// ---- 20_Product/10_BCF/11_Conv/10_Base/F_DeleteDestination.TcPOU
FUNCTION F_DeleteDestination : BOOL
(**************************************************************************************
 * 	Application		:	BoxControl Framework
 *	Revision		:	$Revision: 404529 $
 *	Revision date	:	$Date: 2018-04-23 08:21:38 +0200 (Mo., 23 Apr 2018) $
 *	Last changed by	:	$Author: b7bolm $
 *	URL				:	$URL: http://almscdc.swisslog.com/repo/SWPD/Development/BoxControlFramework/20_Release/trunk/01_Software/BCF/BCF/JumpStart/20_Product/10_App/10_Base/10_Lib/10_Conv/F_DeleteDestination.TcPOU $
 *
 *	Purpose			:	Request to delete a Destination in the TU data of a position.
 *						When the destination gets found - clear all other optional destinations.
 *
 * ------------------------------------------------------------------------------------
 *	Copyright Swisslog [IP AG], Switzerland. All rights reserved.
 * 
 * ------------------------------------------------------------------------------------
 *	
 * 	Revision History: 
 *
 * 	VERSION			DATE			INITIALS			DESCRIPTION
 *	0.1				01.01.2001		swl					Example
 *
 **************************************************************************************)
VAR_INPUT
	eFunctionNumber		: E_FunctionNumber; // Number of the function
	ZoneNumber			: INT; // Number of the zone in the function
END_VAR

VAR
	TU_DataIndex	: DINT; // TU-DataIndex
	Idx	  			: INT; // Index variable
END_VAR

// Initialize
F_DeleteDestination := FALSE;

// Get TU_DataIndex
TU_DataIndex := F_GetTU_DataIndex(
					eFunctionNumber := eFunctionNumber, // Position
					ZoneNumber := ZoneNumber); // Zone

// Check if the destination and the current position matches 
FOR Idx := 1 TO TU_DataTable[TU_DataIndex].DataSet.NumberOfDest DO
	IF TU_DataTable[TU_DataIndex].Destination[Idx].eFunctionNumber = eFunctionNumber
	   AND TU_DataTable[TU_DataIndex].Destination[Idx].ZoneNumber = ZoneNumber THEN
		// Destination found
		F_DeleteDestination := TRUE;
		EXIT;
	END_IF
END_FOR

// Destination was found - Delete all other optional destinations and update job present
IF F_DeleteDestination THEN
	// Clear destination table 
	MEMSET(destAddr := ADR(TU_DataTable[TU_DataIndex].Destination),fillByte := 0, n := SIZEOF(TU_DataTable[TU_DataIndex].Destination));
		
	// Reset number of destinations and reset JobPresent
	TU_DataTable[TU_DataIndex].DataSet.NumberOfDest := 0;
	TU_DataTable[TU_DataIndex].DataSet.JobPresent := FALSE;
END_IF

END_FUNCTION

// ---- 20_Product/10_BCF/11_Conv/11_Com/11_ITC/FB_ITC_ConveyorEmulation.TcPOU
FUNCTION_BLOCK FB_ITC_ConveyorEmulation IMPLEMENTS ITF_ITC_Emulation
(**************************************************************************************
 * 	Application		:	BoxControl Framework
 *	Revision		:	$Revision: 404529 $
 *	Revision date	:	$Date: 2018-04-23 08:21:38 +0200 (Mo., 23 Apr 2018) $
 *	Last changed by	:	$Author: b7bolm $
 *	URL				:	$URL: http://almscdc.swisslog.com/repo/SWPD/Development/BoxControlFramework/20_Release/trunk/01_Software/BCF/BCF/JumpStart/20_Product/11_Emu/11_Com/10_Lib/10_Conv/11_ITC/FB_ITC_CoveyorEmulation.TcPOU $
 *
 *	Purpose			:	ITC - Message Manager emulation.
 *						Represents the interface between the application and the 
 *						communication. Serves as abstract layer to ensure application
 *						independency.
 *
 * ------------------------------------------------------------------------------------
 *	Copyright Swisslog [IP AG], Switzerland. All rights reserved.
 * 
 * ------------------------------------------------------------------------------------
 *	
 * 	Revision History: 
 *
 * 	VERSION			DATE			INITIALS			DESCRIPTION
 *	0.1				01.01.2001		swl					Example
 *
 **************************************************************************************)
VAR
	fbDebugMsg			: FB_DebugMsg; // Debug instance
	DebugMsg			: T_MAXSTRING; // Debug msg
	TelegramPosition	: ST_PositionIdent; // Position
	TelegramElement		: E_ElementNumber; // Element
	TelegramGroup		: E_GroupNumber; // Group
	TelegramSubsystem	: BOOL; // Telegram for Subsystem
	TU_DataIndex		: DINT; // TU Data index
	eMsgType			: E_ITC_MsgTypeConv; // Message type conveyor
	
	Data				: ST_ITC_GeneralData; // General data
END_VAR

;

METHOD M_AddData : BOOL
(**************************************************************************************
 * 	Application		:	BoxControl Framework
 *	Revision		:	$Revision: 404529 $
 *	Revision date	:	$Date: 2018-04-23 08:21:38 +0200 (Mo., 23 Apr 2018) $
 *	Last changed by	:	$Author: b7bolm $
 *	URL				:	$URL: http://almscdc.swisslog.com/repo/SWPD/Development/BoxControlFramework/20_Release/trunk/01_Software/BCF/BCF/JumpStart/20_Product/11_Emu/11_Com/10_Lib/10_Conv/11_ITC/FB_ITC_CoveyorEmulation.TcPOU $
 *
 *	Purpose			:	Add data to the emulation system
 *
 * ------------------------------------------------------------------------------------
 *	Copyright Swisslog [IP AG], Switzerland. All rights reserved.
 * 
 * ------------------------------------------------------------------------------------
 *	
 * 	Revision History: 
 *
 * 	VERSION			DATE			INITIALS			DESCRIPTION
 *	0.1				01.01.2001		swl					Example
 *
 **************************************************************************************)
VAR_INPUT
	meChannelSrc	: E_MFCS_Channel;
	mMsgType		: INT;
	mpData			: PVOID;
	mLen			: UDINT;
END_VAR

// Translate type to enumeration
eMsgType := mMsgType;

// Go to corresponding type
CASE eMsgType OF
	(****************************************************
	  No Message type
	*****************************************************)	
	E_ITC_MsgTypeConv.NO_MESSAGE_TYPE:
		;
		
	(****************************************************
	  Add TU request
	*****************************************************)	
	E_ITC_MsgTypeConv.E_ADD_TU_REQUEST:
		// Process
		M_AddData := M_ProcessATQ(
						meChannelSrc := meChannelSrc,
						mpATQ		 := mpData,
						mLen		 := mLen);
		
	(****************************************************
	  Remove TU request
	*****************************************************)	
	E_ITC_MsgTypeConv.E_REMOVE_TU_REQUEST:
		// Process
		M_AddData := M_ProcessRTQ(
						meChannelSrc := meChannelSrc,
						mpRTQ		 := mpData,
						mLen		 := mLen);
	
	(****************************************************
	  Error request
	*****************************************************)	
	E_ITC_MsgTypeConv.E_ERROR_REQUEST:
		// Process
		M_AddData := M_ProcessERQ(
						meChannelSrc := meChannelSrc,
						mpERQ		 := mpData,
						mLen		 := mLen);
	
ELSE
	// Unknown type
	DebugMsg := 'Unknown message type received';
	fbDebugMsg.M_SendErrorMsg(mMessage := DebugMsg);		
END_CASE
END_METHOD

{attribute 'object_name' := 'M_CallITC_Service'}
METHOD M_CallITC_Service : BOOL
END_METHOD

METHOD PRIVATE M_ProcessATQ : BOOL
(**************************************************************************************
 * 	Application		:	BoxControl Framework
 *	Revision		:	$Revision: 404529 $
 *	Revision date	:	$Date: 2018-04-23 08:21:38 +0200 (Mo., 23 Apr 2018) $
 *	Last changed by	:	$Author: b7bolm $
 *	URL				:	$URL: http://almscdc.swisslog.com/repo/SWPD/Development/BoxControlFramework/20_Release/trunk/01_Software/BCF/BCF/JumpStart/20_Product/11_Emu/11_Com/10_Lib/10_Conv/11_ITC/FB_ITC_CoveyorEmulation.TcPOU $
 *
 *	Purpose			:	Add ATQ
 *
 * ------------------------------------------------------------------------------------
 *	Copyright Swisslog [IP AG], Switzerland. All rights reserved.
 * 
 * ------------------------------------------------------------------------------------
 *	
 * 	Revision History: 
 *
 * 	VERSION			DATE			INITIALS			DESCRIPTION
 *	0.1				01.01.2001		swl					Example
 *
 **************************************************************************************)
VAR_INPUT
	meChannelSrc		: E_MFCS_Channel; // Source communicaton channel
	mpATQ				: POINTER TO ST_ITC_ATQ; // Pointer to ATQ
	mLen				: UDINT; // Data length
END_VAR

VAR
	mrFunction		: REFERENCE TO FB_BaseObjectEmulation;
END_VAR

// Search position in registry
TelegramPosition := F_SearchFunctionPosition(Position := mpATQ^.Position);

// If a position and zone was found
IF TelegramPosition.eFunctionNumber > E_FunctionNumber.F_BEGIN_FUNCTION AND
   TelegramPosition.ZoneNumber > 0 THEN
   
   // Store reference of this position
   mrFunction REF= FunctionRegistryEmulation[TelegramPosition.eFunctionNumber].rFunction;
   
   // Check the reference from this position is valid
   IF __ISVALIDREF(mrFunction) THEN
	   
		// Get Data index from this position
		TU_DataIndex := F_GetTU_DataIndexEmulation(
							eFunctionNumber := TelegramPosition.eFunctionNumber,
							ZoneNumber		:= TelegramPosition.ZoneNumber);
		
		// If no data was found on this position
		IF TU_DataIndex = 0 THEN
			// Create a new set
			TU_DataIndex := F_InsertTU_DataEmulation(
								eFunctionNumber := TelegramPosition.eFunctionNumber,
								ZoneNumber 		:= TelegramPosition.ZoneNumber);
	
			// If a index could be created
			IF TU_DataIndex > 0 THEN
				TU_DataTableEmulation[TU_DataIndex].Label.ASCII := mpATQ^.Label;
				TU_DataTableEmulation[TU_DataIndex].Label.HashCode := F_CreateHashCode(mpATQ^.Label);
				TU_DataTableEmulation[TU_DataIndex].DataSet.Dimension.Weight := mpATQ^.Weight;
				TU_DataTableEmulation[TU_DataIndex].DataSet.Dimension.Length := mpATQ^.Length;
				TU_DataTableEmulation[TU_DataIndex].DataSet.Dimension.Height := mpATQ^.Height;
				TU_DataTableEmulation[TU_DataIndex].DataSet.Dimension.Width := mpATQ^.Width;
				TU_DataTableEmulation[TU_DataIndex].DataSet.LongSideLeading := mpATQ^.LongSideLeading;
				TU_DataTableEmulation[TU_DataIndex].DataSet.DataPresent := TRUE;
				
				// Prepare data
				Data.TU_DataIndex := TU_DataIndex;
				Data.ZoneNumber := TelegramPosition.ZoneNumber;
				
				M_ProcessToFunction(
					meFunctionNumber := TelegramPosition.eFunctionNumber,
					mZoneNumber 	 := TelegramPosition.ZoneNumber,
					meChannelSrc	 := meChannelSrc,
					mMsgType		 := E_ITC_MsgTypeConv.E_ADD_TU_REQUEST,
					mpData			 := ADR(Data),
					mLen			 := SIZEOF(Data));
			END_IF
		
		// Otherwise overwrite current index
		ELSIF TU_DataIndex > 0 THEN
			
			// Overwrite
			TU_DataTableEmulation[TU_DataIndex].Label.ASCII := mpATQ^.Label;
			TU_DataTableEmulation[TU_DataIndex].Label.HashCode := F_CreateHashCode(mpATQ^.Label);
			TU_DataTableEmulation[TU_DataIndex].DataSet.Dimension.Weight := mpATQ^.Weight;
			TU_DataTableEmulation[TU_DataIndex].DataSet.Dimension.Length := mpATQ^.Length;
			TU_DataTableEmulation[TU_DataIndex].DataSet.Dimension.Height := mpATQ^.Height;
			TU_DataTableEmulation[TU_DataIndex].DataSet.Dimension.Width := mpATQ^.Width;
			TU_DataTableEmulation[TU_DataIndex].DataSet.LongSideLeading := mpATQ^.LongSideLeading;
			TU_DataTableEmulation[TU_DataIndex].DataSet.DataPresent := TRUE;
		END_IF
		
		F_ITC_SendATR(
			eChannelSrc  := meChannelSrc, 
			PositionName := mpATQ^.Position, 
			eReturnCode  := E_ErrorConv.NO_ERROR_CODE);
	END_IF

// Unknown destination received 
ELSE
	// debug message: '11-000-0000-00-0,  unknown position addressed,  telegram = ATQ,  Position = 99-999-9999-99-9'
	DebugMsg:= '';
	DebugMsg:= CONCAT(DebugMsg, F_AddDividerToSisString(SubsystemRegistry.SubsystemName));
	DebugMsg:= CONCAT(DebugMsg, ',  unknown position addressed');
	DebugMsg:= CONCAT(DebugMsg, DebugTextBlocks.TELEGRAM);
	DebugMsg:= CONCAT(DebugMsg, 'ATQ');
	DebugMsg:= CONCAT(DebugMsg, DebugTextBlocks.POSITION);
	DebugMsg:= CONCAT(DebugMsg, F_AddDividerToSisString(Name:= mpATQ^.Position)  );
	fbDebugMsg.M_SendErrorMsg(mMessage := DebugMsg);

	// Reject telegram
	F_ITC_SendATR(
		eChannelSrc  := meChannelSrc, 
		PositionName := mpATQ^.Position, 
		eReturnCode  := E_ErrorConv.FUNCTIONNUMBER_UNKNOWN);
END_IF
END_METHOD

METHOD PRIVATE M_ProcessERQ : BOOL
(**************************************************************************************
 * 	Application		:	BoxControl Framework
 *	Revision		:	$Revision: 404529 $
 *	Revision date	:	$Date: 2018-04-23 08:21:38 +0200 (Mo., 23 Apr 2018) $
 *	Last changed by	:	$Author: b7bolm $
 *	URL				:	$URL: http://almscdc.swisslog.com/repo/SWPD/Development/BoxControlFramework/20_Release/trunk/01_Software/BCF/BCF/JumpStart/20_Product/11_Emu/11_Com/10_Lib/10_Conv/11_ITC/FB_ITC_CoveyorEmulation.TcPOU $
 *
 *	Purpose			:	Add ERR
 *
 * ------------------------------------------------------------------------------------
 *	Copyright Swisslog [IP AG], Switzerland. All rights reserved.
 * 
 * ------------------------------------------------------------------------------------
 *	
 * 	Revision History: 
 *
 * 	VERSION			DATE			INITIALS			DESCRIPTION
 *	0.1				01.01.2001		swl					Example
 *
 **************************************************************************************)
VAR_INPUT
	meChannelSrc		: E_MFCS_Channel; // Source communicaton channel
	mpERQ				: POINTER TO ST_ITC_ERQ; // Pointer to ERQ
	mLen				: UDINT; // Data length
END_VAR

// Try to find position in registry
TelegramPosition := F_SearchFunctionPosition(Position := mpERQ^.Position);

// Try to find element in registry
TelegramElement := F_SearchElementPosition(ElementName := mpERQ^.Position);

// Try to find group in registry
TelegramGroup := F_SearchGroupNumber(GroupName := mpERQ^.Position);

// Is it for the Subsystem
TelegramSubsystem := F_EqualSisNames(Name1 := SubsystemRegistry.SubsystemName,
                                     Name2 := mpERQ^.Position);

// If a position was found
IF TelegramPosition.eFunctionNumber > E_FunctionNumber.F_BEGIN_FUNCTION THEN
   
	M_ProcessToFunction(
		meFunctionNumber	:= TelegramPosition.eFunctionNumber, 
		mZoneNumber			:= TelegramPosition.ZoneNumber, 
		meChannelSrc		:= meChannelSrc, 
		mMsgType			:= E_ITC_MsgTypeConv.E_ERROR_REQUEST,
		mpData				:= mpERQ, 
		mLen				:= mLen);

// If a element was found
ELSIF TelegramElement > E_ElementNumber.E_BEGIN_ELEMENT THEN
   
	M_ProcessToElement(
		meElementNumber	:= TelegramElement, 
		meChannelSrc	:= meChannelSrc, 
		mMsgType		:= E_ITC_MsgTypeConv.E_ERROR_REQUEST,
		mpData			:= mpERQ, 
		mLen			:= mLen);

// If a group was found
ELSIF TelegramGroup > E_GroupNumber.G_BEGIN_GROUP THEN
   
	M_ProcessToGroup(
		meGroupNumber	:= TelegramGroup, 
		meChannelSrc	:= meChannelSrc, 
		mMsgType		:= E_ITC_MsgTypeConv.E_ERROR_REQUEST,
		mpData			:= mpERQ, 
		mLen			:= mLen);
		
// If it was for the Subsystem
ELSIF TelegramSubsystem THEN
   
	M_ProcessToSubsystem(
		meChannelSrc	:= meChannelSrc, 
		mMsgType		:= E_ITC_MsgTypeConv.E_ERROR_REQUEST,
		mpData			:= mpERQ, 
		mLen			:= mLen);
   
ELSE
	F_ITC_SendERR(
		eChannelSrc	:= meChannelSrc, 
		PositionName:= mpERQ^.Position, 
		Code		:= mpERQ^.Code, 
		eReturnCode	:= E_ErrorConv.WRONG_VALUE);
		
	// Unknown destination received 
	DebugMsg := CONCAT('M_ProcessERQ, Unknown position in Telegram: ', mpERQ^.Position);
	fbDebugMsg.M_SendErrorMsg(mMessage := DebugMsg);	
END_IF
END_METHOD

METHOD PRIVATE M_ProcessRTQ : BOOL
(**************************************************************************************
 * 	Application		:	BoxControl Framework
 *	Revision		:	$Revision: 404529 $
 *	Revision date	:	$Date: 2018-04-23 08:21:38 +0200 (Mo., 23 Apr 2018) $
 *	Last changed by	:	$Author: b7bolm $
 *	URL				:	$URL: http://almscdc.swisslog.com/repo/SWPD/Development/BoxControlFramework/20_Release/trunk/01_Software/BCF/BCF/JumpStart/20_Product/11_Emu/11_Com/10_Lib/10_Conv/11_ITC/FB_ITC_CoveyorEmulation.TcPOU $
 *
 *	Purpose			:	Add RTQ
 *
 * ------------------------------------------------------------------------------------
 *	Copyright Swisslog [IP AG], Switzerland. All rights reserved.
 * 
 * ------------------------------------------------------------------------------------
 *	
 * 	Revision History: 
 *
 * 	VERSION			DATE			INITIALS			DESCRIPTION
 *	0.1				01.01.2001		swl					Example
 *
 **************************************************************************************)
VAR_INPUT
	meChannelSrc		: E_MFCS_Channel; // Source communicaton channel
	mpRTQ				: POINTER TO ST_ITC_RTQ; // Pointer to RTQ
	mLen				: UDINT; // Data length
END_VAR

// Search position in registry
TelegramPosition := F_SearchFunctionPosition(Position := mpRTQ^.Position);

// If a position and zone was found
IF TelegramPosition.eFunctionNumber > E_FunctionNumber.F_BEGIN_FUNCTION AND
   TelegramPosition.ZoneNumber > 0 THEN
   
	// Prepare data
	Data.ZoneNumber := TelegramPosition.ZoneNumber;
	
	M_ProcessToFunction(
		meFunctionNumber := TelegramPosition.eFunctionNumber,
		mZoneNumber 	 := TelegramPosition.ZoneNumber,
		meChannelSrc	 := meChannelSrc,
		mMsgType		 := E_ITC_MsgTypeConv.E_REMOVE_TU_REQUEST,
		mpData			 := ADR(Data),
		mLen		     := SIZEOF(Data));

ELSE
	// Position not valid
	F_ITC_SendRTR(
		eChannelSrc	:= meChannelSrc, 
		PositionName:= mpRTQ^.Position, 
		eReturnCode	:= E_ErrorConv.WRONG_VALUE);
		
	// Unknown destination received 
	DebugMsg := CONCAT('M_ProcessRTQ, Unknown position in Telegram: ', mpRTQ^.Position);
	fbDebugMsg.M_SendErrorMsg(mMessage := DebugMsg);	
END_IF
END_METHOD

METHOD PRIVATE M_ProcessToElement : BOOL
(**************************************************************************************
 * 	Application		:	BoxControl Framework
 *	Revision		:	$Revision: 404529 $
 *	Revision date	:	$Date: 2018-04-23 08:21:38 +0200 (Mo., 23 Apr 2018) $
 *	Last changed by	:	$Author: b7bolm $
 *	URL				:	$URL: http://almscdc.swisslog.com/repo/SWPD/Development/BoxControlFramework/20_Release/trunk/01_Software/BCF/BCF/JumpStart/20_Product/11_Emu/11_Com/10_Lib/10_Conv/11_ITC/FB_ITC_CoveyorEmulation.TcPOU $
 *
 *	Purpose			:	ITC - Process message to element
 *
 * ------------------------------------------------------------------------------------
 *	Copyright Swisslog [IP AG], Switzerland. All rights reserved.
 * 
 * ------------------------------------------------------------------------------------
 *	
 * 	Revision History: 
 *
 * 	VERSION			DATE			INITIALS			DESCRIPTION
 *	0.1				01.01.2001		swl					Example
 *
 **************************************************************************************)
VAR_INPUT
	meElementNumber	: E_ElementNumber;
	meChannelSrc	: E_MFCS_Channel; // Source communicaton channel
	mMsgType		: INT; // msg type
	mpData			: PVOID; // data pointer
	mLen			: UDINT; // Data length
END_VAR

VAR
	mrefObject		: REFERENCE TO FB_BaseObjectEmulation; // Reference
END_VAR
// Initialize
M_ProcessToElement := TRUE;

// Check if ElementNumber is valid
IF meElementNumber > E_ElementNumber.E_BEGIN_ELEMENT AND 
   meElementNumber < E_ElementNumber.E_END_ELEMENT THEN
	// Set reference
	mrefObject REF= ElementRegistryEmulation[meElementNumber].rElement;
	
	// Check if reference is valid
	IF __ISVALIDREF(mrefObject) THEN
			// Forward message to corresponding object
		M_ProcessToElement := mrefObject.M_ITC_ProcessMsg(
								meChannelSrc := meChannelSrc, 
								mMsgType	 := mMsgType, 
								mpData		 := mpData,
								mLen	     := mLen); 
	END_IF	
END_IF
END_METHOD

METHOD PRIVATE M_ProcessToFunction : BOOL
(**************************************************************************************
 * 	Application		:	BoxControl Framework
 *	Revision		:	$Revision: 404529 $
 *	Revision date	:	$Date: 2018-04-23 08:21:38 +0200 (Mo., 23 Apr 2018) $
 *	Last changed by	:	$Author: b7bolm $
 *	URL				:	$URL: http://almscdc.swisslog.com/repo/SWPD/Development/BoxControlFramework/20_Release/trunk/01_Software/BCF/BCF/JumpStart/20_Product/11_Emu/11_Com/10_Lib/10_Conv/11_ITC/FB_ITC_CoveyorEmulation.TcPOU $
 *
 *	Purpose			:	ITC - Process message to function
 *
 * ------------------------------------------------------------------------------------
 *	Copyright Swisslog [IP AG], Switzerland. All rights reserved.
 * 
 * ------------------------------------------------------------------------------------
 *	
 * 	Revision History: 
 *
 * 	VERSION			DATE			INITIALS			DESCRIPTION
 *	0.1				01.01.2001		swl					Example
 *
 **************************************************************************************)
VAR_INPUT
	meFunctionNumber	: E_FunctionNumber; // Function number
	mZoneNumber			: INT; // Zone number
	meChannelSrc		: E_MFCS_Channel; // Source communicaton channel
	mMsgType		: INT; // msg type
	mpData			: PVOID; // data pointer
	mLen			: UDINT; // Data length
END_VAR

VAR
	mrefObject			: REFERENCE TO FB_BaseObjectEmulation; // Reference
END_VAR
// Initialize
M_ProcessToFunction := TRUE;

// If a valid function was found with a valid zone
IF 	meFunctionNumber > E_FunctionNumber.F_BEGIN_FUNCTION AND 
	meFunctionNumber < E_FunctionNumber.F_END_FUNCTION AND 
	mZoneNumber >= 0 AND mZoneNumber <= NUMBER_OF_ZONES_PER_FUNCTION THEN

	// Set reference 
	mrefObject REF= FunctionRegistryEmulation[meFunctionNumber].rFunction;
	
	// Check if reference is valid
	IF __ISVALIDREF(mrefObject) THEN

		// Call M_ITC_AddToBuffer
		M_ProcessToFunction := mrefObject.M_ITC_ProcessMsg(
								meChannelSrc := meChannelSrc, 
								mMsgType	 := mMsgType, 
								mpData		 := mpData,
								mLen		 := mLen); 
	END_IF
END_IF
END_METHOD

METHOD PRIVATE M_ProcessToGroup : BOOL
(**************************************************************************************
 * 	Application		:	BoxControl Framework
 *	Revision		:	$Revision: 404529 $
 *	Revision date	:	$Date: 2018-04-23 08:21:38 +0200 (Mo., 23 Apr 2018) $
 *	Last changed by	:	$Author: b7bolm $
 *	URL				:	$URL: http://almscdc.swisslog.com/repo/SWPD/Development/BoxControlFramework/20_Release/trunk/01_Software/BCF/BCF/JumpStart/20_Product/11_Emu/11_Com/10_Lib/10_Conv/11_ITC/FB_ITC_CoveyorEmulation.TcPOU $
 *
 *	Purpose			:	ITC - Process message to group
 *
 * ------------------------------------------------------------------------------------
 *	Copyright Swisslog [IP AG], Switzerland. All rights reserved.
 * 
 * ------------------------------------------------------------------------------------
 *	
 * 	Revision History: 
 *
 * 	VERSION			DATE			INITIALS			DESCRIPTION
 *	0.1				01.01.2001		swl					Example
 *
 **************************************************************************************)
VAR_INPUT
	meGroupNumber		: E_GroupNumber; // Groupnumber
	meChannelSrc		: E_MFCS_Channel; // Source communicaton channel
	mMsgType		: INT; // msg type
	mpData			: PVOID; // data pointer
	mLen			: UDINT; // Data length
END_VAR

VAR
	mrefObject			: REFERENCE TO FB_BaseObjectEmulation; // Reference
END_VAR
// Initialize
M_ProcessToGroup := TRUE;

// Check if GroupNumber is valid
IF meGroupNumber > E_GroupNumber.G_BEGIN_GROUP AND 
   meGroupNumber < E_GroupNumber.G_END_GROUP THEN
	// Set reference
	mrefObject REF= GroupRegistryEmulation[meGroupNumber].rGroup;
	
	// Check if reference is valid
	IF __ISVALIDREF(mrefObject) THEN
		
		// Send ITC-message to a specified group
		M_ProcessToGroup := mrefObject.M_ITC_ProcessMsg(
								meChannelSrc := meChannelSrc, 
								mMsgType	 := mMsgType, 
								mpData		 := mpData,
								mLen		 := mLen); 	
	END_IF
END_IF
END_METHOD

METHOD PRIVATE M_ProcessToSubsystem : BOOL
(**************************************************************************************
 * 	Application		:	BoxControl Framework
 *	Revision		:	$Revision: 404529 $
 *	Revision date	:	$Date: 2018-04-23 08:21:38 +0200 (Mo., 23 Apr 2018) $
 *	Last changed by	:	$Author: b7bolm $
 *	URL				:	$URL: http://almscdc.swisslog.com/repo/SWPD/Development/BoxControlFramework/20_Release/trunk/01_Software/BCF/BCF/JumpStart/20_Product/11_Emu/11_Com/10_Lib/10_Conv/11_ITC/FB_ITC_CoveyorEmulation.TcPOU $
 *
 *	Purpose			:	ITC - Process message to subsystem
 *
 * ------------------------------------------------------------------------------------
 *	Copyright Swisslog [IP AG], Switzerland. All rights reserved.
 * 
 * ------------------------------------------------------------------------------------
 *	
 * 	Revision History: 
 *
 * 	VERSION			DATE			INITIALS			DESCRIPTION
 *	0.1				01.01.2001		swl					Example
 *
 **************************************************************************************)
VAR_INPUT
	meChannelSrc		: E_MFCS_Channel; // Source communicaton channel
	mMsgType		: INT; // msg type
	mpData			: PVOID; // data pointer
	mLen			: UDINT; // Data length
END_VAR

VAR
	mrefObject			: REFERENCE TO FB_BaseObjectEmulation; // Reference
END_VAR
// Initialize
M_ProcessToSubsystem := TRUE;

// Set reference 
mrefObject REF= SubsystemRegistryEmulation.rSubsystem;

// Check if reference is valid
IF __ISVALIDREF(mrefObject) THEN
	// Call M_ITC_AddToBuffer
	M_ProcessToSubsystem := mrefObject.M_ITC_ProcessMsg(
								meChannelSrc := meChannelSrc, 
								mMsgType	 := mMsgType, 
								mpData		 := mpData,
								mLen		 := mLen);
END_IF
END_METHOD

END_FUNCTION_BLOCK

// ---- 20_Product/10_BCF/11_Conv/11_Com/11_ITC/F_ITC_SendATR.TcPOU
FUNCTION F_ITC_SendATR : BOOL
(**************************************************************************************
 * 	Application		:	BoxControl Framework
 *	Revision		:	$Revision: 404529 $
 *	Revision date	:	$Date: 2018-04-23 08:21:38 +0200 (Mo., 23 Apr 2018) $
 *	Last changed by	:	$Author: b7bolm $
 *	URL				:	$URL: http://almscdc.swisslog.com/repo/SWPD/Development/BoxControlFramework/20_Release/trunk/01_Software/BCF/BCF/JumpStart/20_Product/10_App/11_Com/10_Lib/10_Conv/11_ITC/F_ITC_SendATR.TcPOU $
 *
 *	Purpose			:	Wrap message - ATR
 *
 * ------------------------------------------------------------------------------------
 *	Copyright Swisslog [IP AG], Switzerland. All rights reserved.
 * 
 * ------------------------------------------------------------------------------------
 *	
 * 	Revision History: 
 *
 * 	VERSION			DATE			INITIALS			DESCRIPTION
 *	0.1				01.01.2001		swl					Example
 *
 **************************************************************************************)
VAR_INPUT
	eChannelSrc		: E_MFCS_Channel; // Source communicaton channel
	PositionName	: STRING(Conveyor.POSITION_STRINGLENGTH); // SIS MM-GGG-EEEE-FF-Z
	eReturnCode		: E_ErrorConv; // Return code
END_VAR
VAR
	ATR				: ST_ITC_ATR; 
END_VAR

// Map values
ATR.Position := PositionName;
ATR.ReturnCode := eReturnCode;

// Forward to ITC
F_ITC_SendATR := fbITC_Manager.M_SendData(
					meChannel	:= eChannelSrc,
					mMsgType	:= E_ITC_MsgTypeConv.E_ADD_TU_REPORT,
					mpData		:= ADR(ATR),
					mLen		:= SIZEOF(ATR));

END_FUNCTION

// ---- 20_Product/10_BCF/11_Conv/11_Com/11_ITC/F_ITC_SendERR.TcPOU
FUNCTION F_ITC_SendERR : BOOL
(**************************************************************************************
 * 	Application		:	BoxControl Framework
 *	Revision		:	$Revision: 404529 $
 *	Revision date	:	$Date: 2018-04-23 08:21:38 +0200 (Mo., 23 Apr 2018) $
 *	Last changed by	:	$Author: b7bolm $
 *	URL				:	$URL: http://almscdc.swisslog.com/repo/SWPD/Development/BoxControlFramework/20_Release/trunk/01_Software/BCF/BCF/JumpStart/20_Product/10_App/11_Com/10_Lib/10_Conv/11_ITC/F_ITC_SendERR.TcPOU $
 *
 *	Purpose			:	Wrap message - ERR
 *
 * ------------------------------------------------------------------------------------
 *	Copyright Swisslog [IP AG], Switzerland. All rights reserved.
 * 
 * ------------------------------------------------------------------------------------
 *	
 * 	Revision History: 
 *
 * 	VERSION			DATE			INITIALS			DESCRIPTION
 *	0.1				01.01.2001		swl					Example
 *
 **************************************************************************************)
VAR_INPUT
	eChannelSrc		: E_MFCS_Channel; // Source communicaton channel
	PositionName	: STRING(Conveyor.POSITION_STRINGLENGTH); // SIS MM-GGG-EEEE-FF-Z
	Code			: INT; // Error type code
	eReturnCode		: E_ErrorConv; // Return code
END_VAR
VAR
	ERR				: ST_ITC_ERR; 
END_VAR

// Map values
ERR.Position := PositionName;
ERR.Code := Code;
ERR.ReturnCode := eReturnCode;

// Forward to ITC
F_ITC_SendERR := fbITC_Manager.M_SendData(
					meChannel	:= eChannelSrc,
					mMsgType	:= E_ITC_MsgTypeConv.E_ERROR_REPORT,
					mpData		:= ADR(ERR),
					mLen		:= SIZEOF(ERR));

END_FUNCTION

// ---- 20_Product/10_BCF/11_Conv/11_Com/11_ITC/F_ITC_SendRTR.TcPOU
FUNCTION F_ITC_SendRTR : BOOL
(**************************************************************************************
 * 	Application		:	BoxControl Framework
 *	Revision		:	$Revision: 404529 $
 *	Revision date	:	$Date: 2018-04-23 08:21:38 +0200 (Mo., 23 Apr 2018) $
 *	Last changed by	:	$Author: b7bolm $
 *	URL				:	$URL: http://almscdc.swisslog.com/repo/SWPD/Development/BoxControlFramework/20_Release/trunk/01_Software/BCF/BCF/JumpStart/20_Product/10_App/11_Com/10_Lib/10_Conv/11_ITC/F_ITC_SendRTR.TcPOU $
 *
 *	Purpose			:	Wrap message - RTR
 *
 * ------------------------------------------------------------------------------------
 *	Copyright Swisslog [IP AG], Switzerland. All rights reserved.
 * 
 * ------------------------------------------------------------------------------------
 *	
 * 	Revision History: 
 *
 * 	VERSION			DATE			INITIALS			DESCRIPTION
 *	0.1				01.01.2001		swl					Example
 *
 **************************************************************************************)
VAR_INPUT
	eChannelSrc		: E_MFCS_Channel; // Source communicaton channel
	PositionName	: STRING(Conveyor.POSITION_STRINGLENGTH); // SIS MM-GGG-EEEE-FF-Z
	eReturnCode		: E_ErrorConv; // Return code
END_VAR
VAR
	RTR				: ST_ITC_RTR; 
END_VAR

// Map values
RTR.Position := PositionName;
RTR.ReturnCode := eReturnCode;

// Forward to ITC
F_ITC_SendRTR := fbITC_Manager.M_SendData(
					meChannel	:= eChannelSrc,
					mMsgType	:= E_ITC_MsgTypeConv.E_REMOVE_TU_REPORT,
					mpData		:= ADR(RTR),
					mLen		:= SIZEOF(RTR));

END_FUNCTION

// ---- 20_Product/20_ProBox/10_Base/09_Overrides/FB_PB_ITC_Conveyor.TcPOU
FUNCTION_BLOCK FB_PB_ITC_Conveyor EXTENDS FB_ITC_Conveyor IMPLEMENTS ITF_ITC 
(**************************************************************************************
 * 	Application		:	BoxControl Framework
 *	Revision		:	$Revision: 417092 $
 *	Revision date	:	$Date: 2018-11-14 12:58:58 +0100 (Mi., 14 Nov 2018) $
 *	Last changed by	:	$Author: q8aberh $
 *	URL				:	$URL: http://almscdc.swisslog.com/repo/SWPD/Development/ProMove/02_Controls/ProBox/03_Implementation/01_DevelopmentProject/01_Software/ProBox_COE/ProBox_DevProj_v1.0/PLC_1/20_Product/10_App/11_Com/10_Lib/10_Conv/11_ITC/FB_ITC_Conveyor.TcPOU $
 *
 *	Purpose			:	ITC - Message Manager.
 *						Represents the interface between the application and the 
 *						communication. Serves as abstract layer to ensure application
 *						independency.
 *
 * ------------------------------------------------------------------------------------
 *	Copyright Swisslog [IP AG], Switzerland. All rights reserved.
 * 
 * ------------------------------------------------------------------------------------
 *	
 * 	Revision History: 
 *
 * 	VERSION			DATE			INITIALS			DESCRIPTION
 *	0.1				01.01.2001		swl					Example
 *
 **************************************************************************************)
VAR_INPUT
	
END_VAR

VAR
	
END_VAR

VAR PERSISTENT
	
END_VAR

(**************************************************************************************************************
   Body never called!
***************************************************************************************************************)
;

METHOD PROTECTED M_ProcessTDQ : BOOL
(**************************************************************************************
 * 	Application		:	BoxControl Framework
 *	Revision		:	$Revision:  $
 *	Revision date	:	$Date: $
 *	Last changed by	:	$Author: q8hedls $
 *	URL				:	$URL: $
 *
 *	Purpose			:	Override BCF process for processing a received Task Delet Request telegram.
 *
 * ------------------------------------------------------------------------------------
 *	Copyright Swisslog [IP AG], Switzerland. All rights reserved.
 * 
 * ------------------------------------------------------------------------------------
 *	
 * 	Revision History: 
 *
 * 	VERSION			DATE			INITIALS			DESCRIPTION
 *	0.1				01.01.2001		swl					Example
 *
 **************************************************************************************)
VAR_INPUT
	meChannelSrc		: E_MFCS_Channel; // Source communicaton channel
	mpTDQ				: POINTER TO ST_ITC_TDQ; // Pointer to TDQ
	mLen				: UDINT; // Data length
END_VAR

VAR
	mPosition 			: ST_PositionIdent ; // Position
END_VAR

// Get position from telegram
mPosition := F_SearchFunctionPosition( Position := mpTDQ^.Position);
IF(mPosition.eFunctionNumber>E_FunctionNumber.F_BEGIN_FUNCTION AND mPosition.ZoneNumber>0) THEN
	F_ResetOccupied(mPosition.eFunctionNumber, mPosition.ZoneNumber);				
END_IF

//proceed with TDQ command
M_ProcessTDQ:= SUPER^.M_ProcessTDQ(meChannelSrc,mpTDQ,mLen);

//Re-initialize the function
IF(mPosition.eFunctionNumber>E_FunctionNumber.F_BEGIN_FUNCTION AND mPosition.ZoneNumber>0) THEN
	F_InitializeFunction(mPosition.eFunctionNumber);
END_IF
END_METHOD

METHOD PROTECTED M_ProcessTTA : BOOL
(**************************************************************************************
 * 	Application		:	BoxControl Framework
 *	Revision		:	$Revision:  $
 *	Revision date	:	$Date: $
 *	Last changed by	:	$Author: q8hedls $
 *	URL				:	$URL: $
 *
 *	Purpose			:	Override BCF process for processing a received Transport Task Assignment telegram.
 *
 * ------------------------------------------------------------------------------------
 *	Copyright Swisslog [IP AG], Switzerland. All rights reserved.
 * 
 * ------------------------------------------------------------------------------------
 *	
 * 	Revision History: 
 *
 * 	VERSION			DATE			INITIALS			DESCRIPTION
 *	0.1				01.01.2001		swl					Example
 *
 **************************************************************************************)
VAR_INPUT
	meChannelSrc		: E_MFCS_Channel; // Source communicaton channel
	mpTTA				: POINTER TO ST_ITC_TTA; // Pointer to TTA
	mLen				: UDINT;
END_VAR

VAR	
	mSensorOccupiedMem	: BOOL; //keep the actual value, to be able to set it back after the call to TTA cmd
	mRestore			: BOOL; //do a restore of SensorOccupied	
END_VAR

// Search position in registry
Position := F_SearchFunctionPosition(Position := mpTTA^.Position);
IF(__ISVALIDREF(F_PB_GetTransportControlDataRef(Position.eFunctionNumber, Position.ZoneNumber))) THEN
	mSensorOccupiedMem := F_PB_GetTransportControlDataRef(Position.eFunctionNumber, Position.ZoneNumber).SensorOccupied;
	mRestore := TRUE;
	IF(F_PB_GetTransportControlDataRef(Position.eFunctionNumber, Position.ZoneNumber).eTakeOverState <> E_TakeOverState.ACTIVE AND
	   F_PB_GetTransportControlDataRef(Position.eFunctionNumber, Position.ZoneNumber).eHandOverState <> E_HandOverState.ACTIVE) THEN
		//For Probox we want to be able to receive TTA despite there are not TU pressent, so we override the SensorOccupied value	   	
		F_PB_GetTransportControlDataRef(Position.eFunctionNumber, Position.ZoneNumber).SensorOccupied := TRUE;
	ELSE
		//force a TTC -> POSITION_NOT_CORRECT_OCCUPIED during an active transport.		
		F_PB_GetTransportControlDataRef(Position.eFunctionNumber, Position.ZoneNumber).SensorOccupied := FALSE;
	END_IF
END_IF
//proceed with TDQ command
M_ProcessTTA:= SUPER^.M_ProcessTTA(meChannelSrc,mpTTA,mLen);

//restore value
IF(mRestore) THEN
	F_PB_GetTransportControlDataRef(Position.eFunctionNumber, Position.ZoneNumber).SensorOccupied := mSensorOccupiedMem;
END_IF
END_METHOD

END_FUNCTION_BLOCK

// ---- 20_Product/20_ProBox/30_Toolbox/F_ResetOccupied.TcPOU
FUNCTION F_ResetOccupied : BOOL
(**************************************************************************************
 * 	Application		:	BoxControl Framework
 *	Revision		:	$Revision: 417092 $
 *	Revision date	:	$Date: 2018-11-14 12:58:58 +0100 (Mi., 14 Nov 2018) $
 *	Last changed by	:	$Author: q8aberh $
 *	URL				:	$URL: http://almscdc.swisslog.com/repo/SWPD/Development/ProMove/02_Controls/ProBox/03_Implementation/01_DevelopmentProject/01_Software/ProBox_COE/ProBox_DevProj_v1.0/PLC_1/20_Product/10_App/12_E_Functions/11_ProBox/02_Functions/F_ResetOccupied.TcPOU $
 *
 *	Purpose			:	Return zone data
 *
 * ------------------------------------------------------------------------------------
 *	Copyright Swisslog [IP AG], Switzerland. All rights reserved.
 * 
 * ------------------------------------------------------------------------------------
 *	
 * 	Revision History: 
 *
 * 	VERSION			DATE			INITIALS			DESCRIPTION
 *	0.1				01.01.2001		swl					Example
 *
 **************************************************************************************)
VAR_INPUT
	eFunctionNumber		: E_FunctionNumber;
	ZoneNumber			: INT; 
END_VAR



// Check if function number and zone is valid
IF eFunctionNumber > E_FunctionNumber.F_BEGIN_FUNCTION AND
   eFunctionNumber < E_FunctionNumber.F_END_FUNCTION AND
   ZoneNumber > 0 AND ZoneNumber <= NUMBER_OF_ZONES_PER_FUNCTION THEN
  
	// Check reference is valid
    IF __ISVALIDREF(FunctionRegistry[eFunctionNumber].rFunction) THEN
	   // Return zone data
	   //FunctionRegistry[eFunctionNumber].rFunction.M_DeleteOccupied(ZoneNumber);
	   IF __ISVALIDREF(FunctionRegistry[eFunctionNumber].Zone[ZoneNumber].refZoneData) THEN
		   FunctionRegistry[eFunctionNumber].Zone[ZoneNumber].refZoneData.TransportControlData.Occupied := FALSE;
		   FunctionRegistry[eFunctionNumber].Zone[ZoneNumber].refZoneData.TransportControlData.NumberOfPresentTUs := 0;
		   F_ResetOccupied := TRUE;
	   END_IF
    END_IF  
END_IF

END_FUNCTION

// ---- 20_Product/10_BCF/11_Conv/12_E_Functions/10_Helper/F_InitializeFunction.TcPOU
FUNCTION F_InitializeFunction :BOOL
(**************************************************************************************
 * 	Application		:	BoxControl Framework
 *	Revision		:	$Revision: 404529 $
 *	Revision date	:	$Date: 2018-04-23 08:21:38 +0200 (Mo., 23 Apr 2018) $
 *	Last changed by	:	$Author: b7bolm $
 *	URL				:	$URL: http://almscdc.swisslog.com/repo/SWPD/Development/BoxControlFramework/20_Release/trunk/01_Software/BCF/BCF/JumpStart/20_Product/10_App/12_E_Functions/10_Lib/10_Conv/10_Functions/F_InitializeFunction.TcPOU $
 *
 *	Purpose			:	Initialize all functions
 *
 * ------------------------------------------------------------------------------------
 *	Copyright Swisslog [IP AG], Switzerland. All rights reserved.
 * 
 * ------------------------------------------------------------------------------------
 *	
 * 	Revision History: 
 *
 * 	VERSION			DATE			INITIALS			DESCRIPTION
 *	0.1				01.01.2001		swl					Example
 *
 **************************************************************************************)
VAR_INPUT
	eFunctionNumber		: E_FunctionNumber; // Function number
END_VAR



// If reference is valid
IF __ISVALIDREF(FunctionRegistry[eFunctionNumber].rFunction) THEN
	// Initialize function
	FunctionRegistry[eFunctionNumber].rFunction.M_InitFunction(TRUE);
END_IF

END_FUNCTION

// ---- 20_Product/20_ProBox/30_Toolbox/F_PB_GetTransportControlDataRef.TcPOU
FUNCTION F_PB_GetTransportControlDataRef : REFERENCE TO ST_TransportControlData
(**************************************************************************************
 * 	Application		:	BoxControl Framework
 *	Revision		:	$Revision:  $
 *	Revision date	:	$Date: $
 *	Last changed by	:	$Author: q8sheds $
 *	URL				:	$URL: $
 *
 *	Purpose			:	return Transport control data as reference
 *
 * ------------------------------------------------------------------------------------
 *	Copyright Swisslog [IP AG], Switzerland. All rights reserved.
 * 
 * ------------------------------------------------------------------------------------
 *	
 * 	Revision History: 
 *
 * 	VERSION			DATE			INITIALS			DESCRIPTION
 *	0.1				01.01.2001		swl					Example
 *
 **************************************************************************************)
VAR_INPUT
	eFunctionNumber		: E_FunctionNumber; // Function number
	ZoneNumber			: INT; // Zone number
END_VAR

//init
F_PB_GetTransportControlDataRef REF= PBTransportCtrl.pbTransportControlDataEmpty;	//return ref to empty transportcontroller data to avoid reutrn of NULL

// Check if function number is valid
IF(  eFunctionNumber > E_FunctionNumber.F_BEGIN_FUNCTION AND eFunctionNumber < E_FunctionNumber.F_END_FUNCTION AND
	 ZoneNumber > 0 AND ZoneNumber <= NUMBER_OF_ZONES_PER_FUNCTION) THEN
	// Check reference is valid
	IF __ISVALIDREF(FunctionRegistry[eFunctionNumber].Zone[ZoneNumber].refZoneData) THEN
   		// Return transport control data   				
		F_PB_GetTransportControlDataRef REF= FunctionRegistry[eFunctionNumber].Zone[ZoneNumber].refZoneData.TransportControlData;
	END_IF
END_IF

END_FUNCTION

// ---- 20_Product/10_BCF/10_Base/10_StateMachine/FB_StateMachine.TcPOU
/// represents a state machine
{attribute 'no_explicit_call' := 'do not call this POU directly'} 
{attribute 'reflection'} 
FUNCTION_BLOCK PUBLIC FB_StateMachine
(**************************************************************************************
 *  Application     :   BoxControl Framework
 *  Revision date   :   $Date: 2021-04-09 08:29:02 +0200 (fre, 09 apr 2021) $
 *  Author          :   CDC
 * ------------------------------------------------------------------------------------
 *  © Swisslog AG
 *  Swisslog is not liable for any usage of this source code that is not agreed 
 *  on between Swisslog and the other party. The mandatory legal liability remains 
 *  unaffected.
 * ------------------------------------------------------------------------------------
 *  Revision History: 
 *
 *  VERSION DATE         INITIALS     DESCRIPTION
 *  0.0     DD.MM.YYYY   (name)       (explain customized modifications)
 *
 **************************************************************************************)
VAR
  {attribute 'instance-path'}
  {attribute 'no_init'}
  Instance          : STRING[255];     // instance path

  SisNbr            : A_InstancePath;  // SIS Number
  Name              : A_InstancePath;  // state machine name
  Tracing           : BOOL  := TRUE;   // HI = state changes are being traced

  State             : UINT;           // current state
  FStateChanged     : BOOL;           // state changed (and new state not yet arrived) 
  TimeStamp         : TIME;           // timestamp of state change
  Duration          : TIME;           // duration of last state

  Callback  : I_StateMachineTextCallback;	// callback event to retrieve state text

  Diagnose  : STRING[255];
END_VAR

VAR_STAT CONSTANT
  REASON_TEXT_LENGTH    : UINT          := 127;
  ARROW                 : STRING[7]     := ' => ';
  MISSING_CALLBACK		: A_StateText   := 'missing StateTextCallback';
END_VAR

METHOD FB_init : BOOL
(**************************************************************************************
 *  Application     :   BoxControl Framework
 *  Revision date   :   $Date: 2021-04-09 08:29:02 +0200 (fre, 09 apr 2021) $
 *  Author          :   CDC
 * ------------------------------------------------------------------------------------
 *  © Swisslog AG
 *  Swisslog is not liable for any usage of this source code that is not agreed 
 *  on between Swisslog and the other party. The mandatory legal liability remains 
 *  unaffected.
 * ------------------------------------------------------------------------------------
 *  Revision History: 
 *
 *  VERSION DATE         INITIALS     DESCRIPTION
 *  0.0     DD.MM.YYYY   (name)       (explain customized modifications)
 *
 **************************************************************************************)
VAR_INPUT
	bInitRetains		: BOOL; // if TRUE, the retain variables are initialized (warm start / cold start)
	bInCopyCode			: BOOL;  // if TRUE, the instance afterwards gets moved into the copy code (online change)

	mName				: A_InstancePath;       		// state machine name
	mStateTextCallback	: I_StateMachineTextCallback;	// callback event to retrieve state text
END_VAR

VAR
	SrcPos  : UINT;
	DstPos  : UINT;
	Length  : UINT;
END_VAR
Name        := mName;
Callback    := mStateTextCallback;

//Remove 'QB2Jumpstart.JumpStart.' from the instance path 
F_InstancePathRemovals(DestStart     := ADR(Instance),
                       DestEnd       := ADR(Instance) + SIZEOF(Instance),
                       RemoveLastPart:= FALSE );
END_METHOD

METHOD PROTECTED M_BuildTraceText
(**************************************************************************************
 *  Application     :   BoxControl Framework
 *  Revision date   :   $Date: 2021-04-09 08:29:02 +0200 (fre, 09 apr 2021) $
 *  Author          :   CDC
 * ------------------------------------------------------------------------------------
 *  © Swisslog AG
 *  Swisslog is not liable for any usage of this source code that is not agreed 
 *  on between Swisslog and the other party. The mandatory legal liability remains 
 *  unaffected.
 * ------------------------------------------------------------------------------------
 *  Revision History: 
 *
 *  VERSION DATE         INITIALS     DESCRIPTION
 *  0.0     DD.MM.YYYY   (name)       (explain customized modifications)
 *
 **************************************************************************************)
VAR_INPUT
  meMsgType       : E_DebugMsgType := E_DebugMsgType.INFO;
  mNewState      : UINT;
  mLastState     : UINT;
  mReason        : POINTER TO BYTE;
END_VAR

VAR
  Trace         : STRING[255];
  LastStateText : A_StateText := MISSING_CALLBACK;
  StateText     : A_StateText := MISSING_CALLBACK;
  DestStart     : POINTER TO BYTE;     // start position to concat
  DestEnd       : POINTER TO BYTE;     // buffer/string end
END_VAR
IF (Tracing = FALSE)
THEN
  RETURN;
END_IF

// get state texts
IF (Callback <> 0)
THEN
  LastStateText:= Callback.M_GetStateText(StateMachine:= THIS, StateNbr:= mLastState );
  StateText    := Callback.M_GetStateText(StateMachine:= THIS, StateNbr:=     P_State );
END_IF

// create trace text
DestStart:= ADR(Trace);
DestEnd  := ADR(Trace) + SIZEOF(Trace);
// sis nbr
DestStart:= F_StringCopy     (DestStart:= DestStart,  DestEnd:= DestEnd,  Source:= ADR(SisNbr)  );

// name
DestStart:= F_StringCopy     (DestStart:= DestStart,  DestEnd:= DestEnd,  Source:= ADR(',  ')  );
DestStart:= F_StringCopy     (DestStart:= DestStart,  DestEnd:= DestEnd,  Source:= ADR(Name)  );
DestStart:= F_StringCopy     (DestStart:= DestStart,  DestEnd:= DestEnd,  Source:= ADR(' changed')  );

// old state
DestStart:= F_StringCopy     (DestStart:= DestStart,  DestEnd:= DestEnd,  Source:= ADR(',  ')  );
DestStart:= F_StringFromUlint(DestStart:= DestStart,  DestEnd:= DestEnd,  Value := mLastState,  Length:= 0  );
DestStart:= F_StringCopy     (DestStart:= DestStart,  DestEnd:= DestEnd,  Source:= ADR(' (')  );
DestStart:= F_StringCopy     (DestStart:= DestStart,  DestEnd:= DestEnd,  Source:= ADR(LastStateText)  );
DestStart:= F_StringCopy     (DestStart:= DestStart,  DestEnd:= DestEnd,  Source:= ADR(')')  );

// new state
DestStart:= F_StringCopy     (DestStart:= DestStart,  DestEnd:= DestEnd,  Source:= ADR(ARROW)  );
DestStart:= F_StringFromUlint(DestStart:= DestStart,  DestEnd:= DestEnd,  Value := State,  Length:= 0  );
DestStart:= F_StringCopy     (DestStart:= DestStart,  DestEnd:= DestEnd,  Source:= ADR(' (')  );
DestStart:= F_StringCopy     (DestStart:= DestStart,  DestEnd:= DestEnd,  Source:= ADR(StateText)  );
DestStart:= F_StringCopy     (DestStart:= DestStart,  DestEnd:= DestEnd,  Source:= ADR(')')  );

// duration
DestStart:= F_StringCopy     (DestStart:= DestStart,  DestEnd:= DestEnd,  Source:= ADR(', duration = ')  );
DestStart:= F_StringFromTime (DestStart:= DestStart,  DestEnd:= DestEnd,  Value := Duration  );

// reason
DestStart:= F_StringCopy     (DestStart:= DestStart,  DestEnd:= DestEnd,  Source:= ADR(', reason = ')  );
DestStart:= F_StringCopy     (DestStart:= DestStart,  DestEnd:= DestEnd,  Source:= mReason  );

// to debug channel
fbDebugMsgManager.M_SendMessage(meMessageType:= meMsgType,
							  mDebugSource := Instance,
							  mpMsgData    := ADR(Trace),
							  mMsgDataLen  := DestStart - ADR(Trace) );

Diagnose:= Trace;
END_METHOD

/// returns the remaining time of state for the given duration
METHOD PUBLIC M_GetRemainingTime : TIME
(**************************************************************************************
 *  Application     :   BoxControl Framework
 *  Revision date   :   $Date: 2021-04-09 08:29:02 +0200 (fre, 09 apr 2021) $
 *  Author          :   CDC
 * ------------------------------------------------------------------------------------
 *  © Swisslog AG
 *  Swisslog is not liable for any usage of this source code that is not agreed 
 *  on between Swisslog and the other party. The mandatory legal liability remains 
 *  unaffected.
 * ------------------------------------------------------------------------------------
 *  Revision History: 
 *
 *  VERSION DATE         INITIALS     DESCRIPTION
 *  0.0     DD.MM.YYYY   (name)       (explain customized modifications)
 *
 **************************************************************************************)
VAR_INPUT
  mDuration  : TIME;    // total duration
END_VAR

VAR
  Remain    : TIME;
END_VAR
IF (P_TimeInState > mDuration)  THEN 
    Remain:= T#0S;
ELSE
    Remain:= mDuration - P_TimeInState;
END_IF

M_GetRemainingTime:= Remain;
END_METHOD

/// re entres the same state with reason
METHOD PUBLIC M_ReEntry
(**************************************************************************************
 *  Application     :   BoxControl Framework
 *  Revision date   :   $Date: 2021-04-09 08:29:02 +0200 (fre, 09 apr 2021) $
 *  Author          :   CDC
 * ------------------------------------------------------------------------------------
 *  © Swisslog AG
 *  Swisslog is not liable for any usage of this source code that is not agreed 
 *  on between Swisslog and the other party. The mandatory legal liability remains 
 *  unaffected.
 * ------------------------------------------------------------------------------------
 *  Revision History: 
 *
 *  VERSION DATE         INITIALS     DESCRIPTION
 *  0.0     DD.MM.YYYY   (name)       (explain customized modifications)
 *
 **************************************************************************************)
VAR_INPUT
  mReason                : STRING[REASON_TEXT_LENGTH]       := '';
END_VAR
FStateChanged:= TRUE;
Duration     := F_GetTimeMsDiff(TimeStamp);
TimeStamp    := F_GetTimeMsTick();


M_BuildTraceText(meMsgType  := E_DebugMsgType.INFO,
                 mNewState := State,
                 mLastState:= State,
                 mReason   := ADR(mReason)  );
END_METHOD

/// sets a new state with reason for change
METHOD PUBLIC M_SetState
(**************************************************************************************
 *  Application     :   BoxControl Framework
 *  Revision date   :   $Date: 2021-04-09 08:29:02 +0200 (fre, 09 apr 2021) $
 *  Author          :   CDC
 * ------------------------------------------------------------------------------------
 *  © Swisslog AG
 *  Swisslog is not liable for any usage of this source code that is not agreed 
 *  on between Swisslog and the other party. The mandatory legal liability remains 
 *  unaffected.
 * ------------------------------------------------------------------------------------
 *  Revision History: 
 *
 *  VERSION DATE         INITIALS     DESCRIPTION
 *  0.0     DD.MM.YYYY   (name)       (explain customized modifications)
 *
 **************************************************************************************)
VAR_INPUT
  mState     : UINT;
  mReason    : STRING[REASON_TEXT_LENGTH];
END_VAR

VAR
  LastState : UINT;
END_VAR
IF State = mState
THEN
  RETURN;
END_IF

LastState:= State;
State   :=  mState;

FStateChanged:= TRUE;
Duration     := F_GetTimeMsDiff(TimeStamp);
TimeStamp    := F_GetTimeMsTick();


M_BuildTraceText(meMsgType  := E_DebugMsgType.INFO,
                 mNewState := State,
                 mLastState:= LastState,
                 mReason   := ADR(mReason)  );
END_METHOD

/// sets a new state with reason for change and severity
METHOD PUBLIC M_SetState1
(**************************************************************************************
 *  Application     :   BoxControl Framework
 *  Revision date   :   $Date: 2021-04-09 08:29:02 +0200 (fre, 09 apr 2021) $
 *  Author          :   CDC
 * ------------------------------------------------------------------------------------
 *  © Swisslog AG
 *  Swisslog is not liable for any usage of this source code that is not agreed 
 *  on between Swisslog and the other party. The mandatory legal liability remains 
 *  unaffected.
 * ------------------------------------------------------------------------------------
 *  Revision History: 
 *
 *  VERSION DATE         INITIALS     DESCRIPTION
 *  0.0     DD.MM.YYYY   (name)       (explain customized modifications)
 *
 **************************************************************************************)
VAR_INPUT
  mMsgType   : E_DebugMsgType := E_DebugMsgType.INFO;
  mState     : UINT;
  mReason    : STRING[REASON_TEXT_LENGTH];
END_VAR

VAR
  LastState : UINT;
END_VAR
IF State = mState
THEN
  RETURN;
END_IF

LastState:= State;
State   :=  mState;

FStateChanged:= TRUE;
Duration     := F_GetTimeMsDiff(TimeStamp);
TimeStamp    := F_GetTimeMsTick();


M_BuildTraceText(meMsgType  := mMsgType,
                 mNewState := State,
                 mLastState:= LastState,
                 mReason   := ADR(mReason)  );
END_METHOD

// entry into new state (must be checked)
//{attribute 'monitoring' := 'call'} no call here
PROPERTY PUBLIC P_Entering : BOOL
GET

(**************************************************************************************************************)
(**************************************************************************************************************)
IF ( FStateChanged = FALSE )
THEN
  P_Entering:= FALSE;
  RETURN;
END_IF




(**************************************************************************************************************)
(**************************************************************************************************************)
FStateChanged:= FALSE;




(**************************************************************************************************************)
(** done ******************************************************************************************************)
P_Entering := TRUE;
END_GET
END_PROPERTY

// exit from old state (optionally)
{attribute 'monitoring' := 'call'}
PROPERTY PUBLIC P_Exiting : BOOL
GET
P_Exiting:= FStateChanged;
END_GET
END_PROPERTY

// SisNbr to trace
{attribute 'monitoring' := 'call'}
PROPERTY PUBLIC P_SisNbr : A_InstancePath
GET
P_SisNbr:= SisNbr;
END_GET
SET
SisNbr:= P_SisNbr;
END_SET
END_PROPERTY

// current state as UINT
{attribute 'monitoring' := 'call'}
PROPERTY PUBLIC P_State : UINT
GET
P_State:= State;
END_GET
END_PROPERTY

// duration of this state
{attribute 'monitoring' := 'call'}
PROPERTY PUBLIC P_TimeInState : TIME
GET
P_TimeInState:= F_GetTimeMsDiff( TimeStamp );
END_GET
END_PROPERTY

// HI = state changes are being traced
{attribute 'monitoring' := 'call'}
PROPERTY PUBLIC P_Tracing : BOOL
GET
P_Tracing:= Tracing;
END_GET
SET
Tracing:= P_Tracing;
END_SET
END_PROPERTY

END_FUNCTION_BLOCK

// ---- 20_Product/10_BCF/10_Base/11_Com/01_Stringhandling/F_StringFromUlint.TcPOU
// converts word to string with specific length (adds zeros)
FUNCTION PUBLIC F_StringFromUlint : POINTER TO BYTE

(**************************************************************************************
 * 	Application		:	BoxControl Framework
 *	Revision		  :	$Revision: 461868 $
 *	Revision date	:	$Date: 1979-01-09 14:35:13 +0200 (Di., 09 Jan 1979) $
 *	Last changed by	:	$Author: b7lipim $
 *	URL				:	$URL: http://almscdc.swisslog.com/repo/SWPD/Development/BoxControlFramework/20_Release/branches/R1.x/01_Software/BCF/BCF/JumpStart/20_Product/10_BCF/10_Base/11_Com/12_DebugMsg/00_GVLs/DebugTextBlocks.TcGVL $
 *
 * ------------------------------------------------------------------------------------
 *	Copyright Swisslog [IP AG], Switzerland. All rights reserved.
 * 
 * ------------------------------------------------------------------------------------
 *	
 * 	Revision History: 
 *
 * VERSION DATE         INITIALS     DESCRIPTION
 * 0.0     DD.MM.YYYY   (name)       (explain customized modifications)
 *
 **************************************************************************************)

(********************************************************************************************************************************)
VAR_INPUT
  DestStart             : POINTER TO BYTE                  := 0;     // = ADR(MyString)                    -> start position to concat
  DestEnd               : POINTER TO BYTE                  := 0;     // = ADR(MyString) + SIZEOF(MyString) -> buffer/string end
  (*----------------------------------------------------------------------------------------------------------------------------*)
  Value                 : ULINT                            := 0;     // value to convert
  Length                : BYTE                             := 0;     // minimum string length (may be left stuffed with zeros)
END_VAR

(********************************************************************************************************************************)
VAR
  DestWork              : POINTER TO BYTE                  := 0;
  (*----------------------------------------------------------------------------------------------------------------------------*)
  Result                : STRING[63]                       := '';
  Size                  : WORD                             := 0;
  Stuff                 : WORD                             := 0;
END_VAR


(********************************************************************************************************************************)
(** check inputs ****************************************************************************************************************)
IF   (DestStart = 0)         THEN  F_StringFromUlint:= 0;          RETURN;
ELSIF(DestEnd   = 0)         THEN  F_StringFromUlint:= DestStart;  RETURN;
ELSIF(DestStart >= DestEnd)  THEN  F_StringFromUlint:= DestStart;  RETURN;
END_IF

DestWork:= DestStart;




(********************************************************************************************************************************)
(** convert *********************************************************************************************************************)
Result:= ULINT_TO_STRING(Value);
Size  := INT_TO_WORD( LEN(Result) );




(********************************************************************************************************************************)
(** stuff? **********************************************************************************************************************)
IF (Size < Length)
THEN
  Stuff:= Length - Size;
  (*-----------------------------------------------------------------*)
  WHILE(Stuff > 0)
  DO
    Stuff:= Stuff - 1;
    (*-------------------------------------------*)
    IF (DestWork >= DestEnd)
    THEN
      DestWork := DestEnd - SIZEOF(DestWork^); // _DestWork^ hier benutzen
      DestWork^:= 16#00;
      DestWork := DestEnd;
      EXIT;
    END_IF
    (*-- add '0' --------------------------------*)
    DestWork^:= 16#30;
    DestWork := DestWork + SIZEOF(DestWork^);
  END_WHILE
END_IF




(********************************************************************************************************************************)
(** copy characters *************************************************************************************************************)
DestWork:= F_StringCopy( DestStart:= DestWork,
                         DestEnd  := DestEnd,
                         Source   := ADR(Result)  );




(********************************************************************************************************************************)
(** done ************************************************************************************************************************)
F_StringFromUlint:= DestWork;

END_FUNCTION

// ---- 20_Product/10_BCF/10_Base/11_Com/01_Stringhandling/F_StringFromTime.TcPOU
// converts word to string with specific length (adds zeros)
FUNCTION PUBLIC F_StringFromTime : POINTER TO BYTE

(**************************************************************************************
 * 	Application		:	BoxControl Framework
 *	Revision		  :	$Revision: 461868 $
 *	Revision date	:	$Date: 1979-01-09 14:35:13 +0200 (Di., 09 Jan 1979) $
 *	Last changed by	:	$Author: b7lipim $
 *	URL				:	$URL: http://almscdc.swisslog.com/repo/SWPD/Development/BoxControlFramework/20_Release/branches/R1.x/01_Software/BCF/BCF/JumpStart/20_Product/10_BCF/10_Base/11_Com/12_DebugMsg/00_GVLs/DebugTextBlocks.TcGVL $
 *
 * ------------------------------------------------------------------------------------
 *	Copyright Swisslog [IP AG], Switzerland. All rights reserved.
 * 
 * ------------------------------------------------------------------------------------
 *	
 * 	Revision History: 
 *
 * VERSION DATE         INITIALS     DESCRIPTION
 * 0.0     DD.MM.YYYY   (name)       (explain customized modifications)
 *
 **************************************************************************************)

(********************************************************************************************************************************)
VAR_INPUT
  DestStart             : POINTER TO BYTE                  := 0;     // = ADR(MyString)                    -> start position to concat
  DestEnd               : POINTER TO BYTE                  := 0;     // = ADR(MyString) + SIZEOF(MyString) -> buffer/string end
  (*----------------------------------------------------------------------------------------------------------------------------*)
  Value                 : TIME                             := T#0S;  // value to convert
END_VAR

(********************************************************************************************************************************)
VAR
  DestWork              : POINTER TO BYTE                  := 0;
  (*----------------------------------------------------------------------------------------------------------------------------*)
  Result                : STRING[15]                       := '';
END_VAR


(********************************************************************************************************************************)
(** check inputs ****************************************************************************************************************)
IF   (DestStart = 0)         THEN  F_StringFromTime:= 0;          RETURN;
ELSIF(DestEnd   = 0)         THEN  F_StringFromTime:= DestStart;  RETURN;
ELSIF(DestStart >= DestEnd)  THEN  F_StringFromTime:= DestStart;  RETURN;
END_IF

DestWork:= DestStart;




(********************************************************************************************************************************)
(** convert *********************************************************************************************************************)
Result:= TIME_TO_STRING(Value);




(********************************************************************************************************************************)
(** copy characters *************************************************************************************************************)
DestWork:= F_StringCopy( DestStart:= DestWork,
                         DestEnd  := DestEnd,
                         Source   := ADR(Result)  );




(********************************************************************************************************************************)
(** done ************************************************************************************************************************)
F_StringFromTime:= DestWork;

END_FUNCTION

// ---- 20_Product/10_BCF/10_Base/11_Com/02_Timings/F_GetBlinkCycle.TcPOU
// returns synchronized blinking pulses with requested (discreet) frequency
FUNCTION PUBLIC F_GetBlinkCycle : BOOL

(**************************************************************************************
 * 	Application		:	BoxControl Framework
 *	Revision		  :	$Revision: 461868 $
 *	Revision date	:	$Date: 1979-01-09 14:35:13 +0200 (Di., 09 Jan 1979) $
 *	Last changed by	:	$Author: b7lipim $
 *	URL				:	$URL: http://almscdc.swisslog.com/repo/SWPD/Development/BoxControlFramework/20_Release/branches/R1.x/01_Software/BCF/BCF/JumpStart/20_Product/10_BCF/10_Base/11_Com/12_DebugMsg/00_GVLs/DebugTextBlocks.TcGVL $
 *
 * ------------------------------------------------------------------------------------
 *	Copyright Swisslog [IP AG], Switzerland. All rights reserved.
 * 
 * ------------------------------------------------------------------------------------
 *	
 * 	Revision History: 
 *
 * VERSION DATE         INITIALS     DESCRIPTION
 * 0.0     DD.MM.YYYY   (name)       (explain customized modifications)
 *
 **************************************************************************************)

(************************************************************************************************************)
VAR_INPUT
  BlinkFrequency        : E_BlinkFrequencies               := E_BlinkFrequencies.Off;
END_VAR

(************************************************************************************************************)
VAR
  {attribute 'displaymode':='hex'}  _TimeTick    : DWORD   := 0;
  {attribute 'displaymode':='hex'}  _TimeMask    : DWORD   := 0;
END_VAR


(********************************************************************************************************************************)
(** calculate *******************************************************************************************************************)
_TimeTick:= TIME_TO_DWORD( TIME() );
_TimeMask:= ( BlinkFrequency AND _TimeTick );




(********************************************************************************************************************************)
(** done ************************************************************************************************************************)
F_GetBlinkCycle:= ( _TimeMask <> 0 );

END_FUNCTION

// ---- 20_Product/10_BCF/10_Base/11_Com/02_Timings/F_GetTimeRemain.TcPOU
// returns remaining time from a timestamp to specified duration
FUNCTION PUBLIC F_GetTimeRemain : TIME

(**************************************************************************************
 * 	Application		:	BoxControl Framework
 *	Revision		  :	$Revision: 461868 $
 *	Revision date	:	$Date: 1979-01-09 14:35:13 +0200 (Di., 09 Jan 1979) $
 *	Last changed by	:	$Author: b7lipim $
 *	URL				:	$URL: http://almscdc.swisslog.com/repo/SWPD/Development/BoxControlFramework/20_Release/branches/R1.x/01_Software/BCF/BCF/JumpStart/20_Product/10_BCF/10_Base/11_Com/12_DebugMsg/00_GVLs/DebugTextBlocks.TcGVL $
 *
 * ------------------------------------------------------------------------------------
 *	Copyright Swisslog [IP AG], Switzerland. All rights reserved.
 * 
 * ------------------------------------------------------------------------------------
 *	
 * 	Revision History: 
 *
 * VERSION DATE         INITIALS     DESCRIPTION
 * 0.0     DD.MM.YYYY   (name)       (explain customized modifications)
 *
 **************************************************************************************)

(********************************************************************************************************************************)
VAR_INPUT
  Duration              : TIME                             := T#0S;    // total duration
  Timestamp             : TIME                             := T#0S;    // time stamp when started
END_VAR

(********************************************************************************************************************************)
VAR
  Elapsed               : TIME                             := T#0S;
  Remain                : TIME                             := T#0S;
END_VAR


(********************************************************************************************************************************)
(** calculate *******************************************************************************************************************)
Elapsed:= F_GetTimeMsDiff(Timestamp);

IF (Elapsed > Duration)  THEN  Remain:= T#0S;
ELSE                           Remain:= Duration - Elapsed;
END_IF



(********************************************************************************************************************************)
(** done ************************************************************************************************************************)
F_GetTimeRemain:= Remain;

END_FUNCTION

// ---- 20_Product/10_BCF/10_Base/F_MemStringReplace.TcPOU
FUNCTION F_MemStringReplace : BOOL
(**************************************************************************************
 * 	Application		:	BoxControl Framework
 *	Revision		:	$Revision: 404529 $
 *	Revision date	:	$Date: 2018-04-23 08:21:38 +0200 (Mo., 23 Apr 2018) $
 *	Last changed by	:	$Author: b7bolm $
 *	URL				:	$URL: http://almscdc.swisslog.com/repo/SWPD/Development/BoxControlFramework/20_Release/trunk/01_Software/BCF/BCF/JumpStart/20_Product/10_App/10_Base/10_Lib/F_MemStringReplace.TcPOU $
 *
 *	Purpose			:	Search in a pointer based structure for a find string, replace 
 *						it with replacement string. If replacement string is shorter, 
 *						move data to close the gap and clean last digits after movement.
 *
 *
 * ------------------------------------------------------------------------------------
 *	Copyright Swisslog [IP AG], Switzerland. All rights reserved.
 * 
 * ------------------------------------------------------------------------------------
 *	
 * 	Revision History: 
 *
 * 	VERSION			DATE			INITIALS			DESCRIPTION
 *	0.1				01.01.2001		swl					Example
 *
 **************************************************************************************)
VAR_INPUT
	pSrc 			: PVOID; // Pointer to source
	FindString		: STRING(MAX_DIGITS); // Find string
	Replacement 	: STRING(MAX_DIGITS); // Replacement string
END_VAR
VAR_IN_OUT
	SrcLen 			: UDINT; // Length of source structure
END_VAR
VAR
	Idx 			: UDINT; // Iterator
	ReplacmentLen 	: UDINT; // Length of string
	FindLen			: UDINT; // Length of string
	RelativeSrc		: UDINT; // Relative source pointer to close gap in data
	RelativeDest	: UDINT; // Relative destination pointer to close gap in data
	pFirstDataByte 	: POINTER TO BYTE; // Pointer to a byte
	pFirstFindByte	: POINTER TO BYTE; // Pointer to a byte
	byte1 			: BYTE;
	byte2			: BYTE;
END_VAR

VAR CONSTANT
	MAX_DIGITS : UDINT := 10; // Max Digits of strings
END_VAR

(* 
Validate Inputs

Length of replacement needs to have the same or a smaller length,
compared to find. Otherwise it would be possible to move data to
the outside of the allocated memory.

*)
IF LEN(Replacement) > LEN(FindString) OR
   pSrc = 0 OR
   SrcLen = 0 THEN
    // Invalid, cancel
	F_MemStringReplace := FALSE;
	RETURN;
END_IF

// Get compare length
ReplacmentLen := INT_TO_UDINT(LEN(Replacement));
FindLen := INT_TO_UDINT(LEN(FindString));

FOR Idx := 0 TO SrcLen - FindLen DO

	pFirstDataByte := pSrc;
	pFirstDataByte := pFirstDataByte + Idx;
	pFirstFindByte := ADR(FindString);
	
	IF (USINT_TO_BYTE(pFirstDataByte^) AND pFirstFindByte^) = pFirstFindByte^ THEN
		(*
		Go through data and compare TO <Find>
		
			0,		Equal
			1/-1, 	Unequal
			0xFF, 	Incorrect parameters
		
		Example:  ABCDEF123GHIJ
				  Find: 123 -> Len : 3
				  Compare ABC with 123
				  Compare BCD with 123
				  Compare CDE with 123
				  ...
		*)		
		IF MEMCMP(pSrc + Idx, ADR(FindString),FindLen) = 0 THEN
			// Replace find with replacement
			MEMCPY(pSrc + Idx, ADR(Replacement), ReplacmentLen);
			
			// If replacement length is smaller than find length, 
			// move data to close the gap
			IF ReplacmentLen < FindLen THEN
				// Build relative addresses
				RelativeSrc := Idx + FindLen;
				RelativeDest := Idx + ReplacmentLen;
				
				(* 
					Example:
					Original:  ABCDEFG   Find BCD, Replacement 12
					Replaced:  A12DEFG
					
					Relativ pointers:   A12DEFG
										   ^^
										   || Source after data
							 Dest for move | 
				*)
				// Check that address is in range of structure
				IF RelativeSrc <= SrcLen THEN
					// Move data to close gap
					MEMCPY(pSrc + RelativeDest, pSrc + RelativeSrc, SrcLen - Idx - FindLen);
					(*
						Example: Moved: A12EFGG
					*)
				END_IF
				
				// Clean unused bytes at the end
				MEMSET(pSrc + SrcLen - FindLen + ReplacmentLen, 0, FindLen - ReplacmentLen);
				// Correction of new length
				SrcLen := SrcLen - FindLen + ReplacmentLen;
				
				(* 
					Example: Cleaned : A12EFG0
				*)
				// Check border
				IF SrcLen < 0 THEN
					SrcLen := 0;
				END_IF
			END_IF
		END_IF
	END_IF
END_FOR

// Return
F_MemStringReplace := TRUE;

END_FUNCTION

// ---- 20_Product/10_BCF/11_Conv/11_Com/11_ITC/F_ITC_SendECR.TcPOU
FUNCTION F_ITC_SendECR : BOOL
(**************************************************************************************
 * 	Application		:	BoxControl Framework
 *	Revision		:	$Revision: 404529 $
 *	Revision date	:	$Date: 2018-04-23 08:21:38 +0200 (Mo., 23 Apr 2018) $
 *	Last changed by	:	$Author: b7bolm $
 *	URL				:	$URL: http://almscdc.swisslog.com/repo/SWPD/Development/BoxControlFramework/20_Release/trunk/01_Software/BCF/BCF/JumpStart/20_Product/10_App/11_Com/10_Lib/10_Conv/11_ITC/F_ITC_SendECR.TcPOU $
 *
 *	Purpose			:	Wrap message - ECR
 *
 * ------------------------------------------------------------------------------------
 *	Copyright Swisslog [IP AG], Switzerland. All rights reserved.
 * 
 * ------------------------------------------------------------------------------------
 *	
 * 	Revision History: 
 *
 * 	VERSION			DATE			INITIALS			DESCRIPTION
 *	0.1				01.01.2001		swl					Example
 *
 **************************************************************************************)
VAR_INPUT
	eChannelSrc		: E_MFCS_Channel; // Source communicaton channel	
	ElementName		: STRING(Conveyor.POSITION_STRINGLENGTH); // The conveyor element which reports its status
	Code			: INT; // ControlCode
	Variable		: DINT; // Variable
	eReturnCode		: E_ErrorConv; // Return code
END_VAR
VAR
	ECR				: ST_ITC_ECR; 
END_VAR

// Map values
ECR.Position := ElementName;
ECR.Code := Code;
ECR.Variable := Variable;
ECR.ReturnCode := eReturnCode;

// Forward to ITC
F_ITC_SendECR := fbITC_Manager.M_SendData(
					meChannel	:= eChannelSrc,
					mMsgType	:= E_ITC_MsgTypeConv.ELEMENT_CONTROL_REPLY,
					mpData		:= ADR(ECR),
					mLen		:= SIZEOF(ECR));

END_FUNCTION

// ---- 20_Product/10_BCF/11_Conv/11_Com/11_ITC/F_ITC_SendESR.TcPOU
FUNCTION F_ITC_SendESR : BOOL
(**************************************************************************************
 * 	Application		:	BoxControl Framework
 *	Revision		:	$Revision: 404529 $
 *	Revision date	:	$Date: 2018-04-23 08:21:38 +0200 (Mo., 23 Apr 2018) $
 *	Last changed by	:	$Author: b7bolm $
 *	URL				:	$URL: http://almscdc.swisslog.com/repo/SWPD/Development/BoxControlFramework/20_Release/trunk/01_Software/BCF/BCF/JumpStart/20_Product/10_App/11_Com/10_Lib/10_Conv/11_ITC/F_ITC_SendESR.TcPOU $
 *
 *	Purpose			:	Wrap message - ESR
 *
 * ------------------------------------------------------------------------------------
 *	Copyright Swisslog [IP AG], Switzerland. All rights reserved.
 * 
 * ------------------------------------------------------------------------------------
 *	
 * 	Revision History: 
 *
 * 	VERSION			DATE			INITIALS			DESCRIPTION
 *	0.1				01.01.2001		swl					Example
 *
 **************************************************************************************)
VAR_INPUT
	eChannelSrc			: E_MFCS_Channel; // Source communicaton channel		
	ElementName	 		: STRING(Conveyor.POSITION_STRINGLENGTH); // SIS MM-GGG-EEEE-FF-Z
	eState				: E_PositionState; // State
	Enabled				: BOOL; // State
	eErrorState			: E_ErrorState; // Error State
	eErrorCode			: E_ErrorConv; // Return Code
	eErrorType			: E_ErrorType; // Error Type
	ErrorInformation	: STRING(System.ERROR_PARAM_STRINGLENGTH); // 5 Chars Error Information
	Variable			: DINT; // Variable
	eReturnCode			: E_ErrorConv; // Return code
END_VAR
VAR
	ESR					: ST_ITC_ESR; 
END_VAR

// Map values
ESR.Position := ElementName;
ESR.Enabled := Enabled;
ESR.State := eState;
ESR.Variable := Variable;
ESR.ErrorCode := eErrorCode;
ESR.ErrorInformation := ErrorInformation;
ESR.ErrorState := eErrorState;
ESR.ErrorType := eErrorType;
ESR.ReturnCode := eReturnCode;

// Forward to ITC
F_ITC_SendESR := fbITC_Manager.M_SendData(
					meChannel	:= eChannelSrc,
					mMsgType	:= E_ITC_MsgTypeConv.ELEMENT_STATUS_REPORT,
					mpData		:= ADR(ESR),
					mLen		:= SIZEOF(ESR));

END_FUNCTION

// ---- 20_Product/10_BCF/11_Conv/11_Com/11_ITC/F_ITC_SendFCR.TcPOU
FUNCTION F_ITC_SendFCR : BOOL
(**************************************************************************************
 * 	Application		:	BoxControl Framework
 *	Revision		:	$Revision: 404529 $
 *	Revision date	:	$Date: 2018-04-23 08:21:38 +0200 (Mo., 23 Apr 2018) $
 *	Last changed by	:	$Author: b7bolm $
 *	URL				:	$URL: http://almscdc.swisslog.com/repo/SWPD/Development/BoxControlFramework/20_Release/trunk/01_Software/BCF/BCF/JumpStart/20_Product/10_App/11_Com/10_Lib/10_Conv/11_ITC/F_ITC_SendFCR.TcPOU $
 *
 *	Purpose			:	Wrap message - FCR
 *
 * ------------------------------------------------------------------------------------
 *	Copyright Swisslog [IP AG], Switzerland. All rights reserved.
 * 
 * ------------------------------------------------------------------------------------
 *	
 * 	Revision History: 
 *
 * 	VERSION			DATE			INITIALS			DESCRIPTION
 *	0.1				01.01.2001		swl					Example
 *
 **************************************************************************************)
VAR_INPUT
	eChannelSrc		: E_MFCS_Channel; // Source communicaton channel	
	FunctionName	: STRING(Conveyor.POSITION_STRINGLENGTH); // The conveyor element which reports its status
	Code			: INT; // ControlCode
	Variable		: DINT; // Variable
	eReturnCode		: E_ErrorConv; // Return code
END_VAR
VAR
	FCR					: ST_ITC_FCR; 
END_VAR

// Map values
FCR.Position := FunctionName;
FCR.Code := Code;
FCR.Variable := Variable;
FCR.ReturnCode := eReturnCode;

// Forward to ITC
F_ITC_SendFCR := fbITC_Manager.M_SendData(
					meChannel	:= eChannelSrc,
					mMsgType	:= E_ITC_MsgTypeConv.FUNCTION_CONTROL_REPLY,
					mpData		:= ADR(FCR),
					mLen		:= SIZEOF(FCR));

END_FUNCTION

// ---- 20_Product/10_BCF/11_Conv/11_Com/11_ITC/F_ITC_SendFSR.TcPOU
FUNCTION F_ITC_SendFSR : BOOL
(**************************************************************************************
 * 	Application		:	BoxControl Framework
 *	Revision		:	$Revision: 404529 $
 *	Revision date	:	$Date: 2018-04-23 08:21:38 +0200 (Mo., 23 Apr 2018) $
 *	Last changed by	:	$Author: b7bolm $
 *	URL				:	$URL: http://almscdc.swisslog.com/repo/SWPD/Development/BoxControlFramework/20_Release/trunk/01_Software/BCF/BCF/JumpStart/20_Product/10_App/11_Com/10_Lib/10_Conv/11_ITC/F_ITC_SendFSR.TcPOU $
 *
 *	Purpose			:	Wrap message - FSR
 *
 * ------------------------------------------------------------------------------------
 *	Copyright Swisslog [IP AG], Switzerland. All rights reserved.
 * 
 * ------------------------------------------------------------------------------------
 *	
 * 	Revision History: 
 *
 * 	VERSION			DATE			INITIALS			DESCRIPTION
 *	0.1				01.01.2001		swl					Example
 *
 **************************************************************************************)
VAR_INPUT
	eChannelSrc			: E_MFCS_Channel; // Source communicaton channel	
	FunctionName		: STRING(Conveyor.POSITION_STRINGLENGTH); // SIS MM-GGG-EEEE-FF-Z
	PrevFunctionNo		: STRING(Conveyor.POSITION_STRINGLENGTH); // SIS MM-GGG-EEEE-FF-Z
	NextFunctionNo		: STRING(Conveyor.POSITION_STRINGLENGTH); // SIS MM-GGG-EEEE-FF-Z
	eState				: E_PositionState; // State
	Enabled				: BOOL; // Enabled
	TransportState		: E_TransportState;
	TakeOverState		: E_TakeOverState;
	HandOverState		: E_HandOverState;
	TU_ID				: STRING(18); // 18 Digit SSID
	TU_Type				: INT; // TU Type
	AssignmentID		: UDINT; // Assignment ID
	LoadInformation		: INT; // 1 = Loaded, 0 = Not loaded
	Destination			: STRING(Conveyor.POSITION_STRINGLENGTH);
	eErrorState			: E_ErrorState; // Error State
	eErrorCode			: E_ErrorConv; // Return Code
	eErrorType			: E_ErrorType; // Error Type
	ErrorInformation	: STRING(System.ERROR_PARAM_STRINGLENGTH); // 5 Chars Error Information
	Variable			: DINT; // Variable
	eReturnCode			: E_ErrorConv; // Return code
END_VAR
VAR
	FSR					: ST_ITC_FSR; 
END_VAR

// Map values
FSR.Position			:= FunctionName;
FSR.PrevFunctionNo		:= PrevFunctionNo;
FSR.NextFunctionNo		:= NextFunctionNo;
FSR.eState				:= eState;
FSR.Enabled				:= Enabled;
FSR.TransportState		:= TransportState;
FSR.TakeOverState		:= TakeOverState;
FSR.HandOverState		:= HandOverState;
FSR.TU_ID				:= TU_ID;
FSR.TU_Type				:= TU_Type;
FSR.AssignmentID		:= AssignmentID;
FSR.LoadInformation		:= LoadInformation;
FSR.Destination			:= Destination;
FSR.eErrorState			:= eErrorState;
FSR.eErrorCode			:= eErrorCode;
FSR.eErrorType			:= eErrorType;
FSR.ErrorInformation	:= ErrorInformation;
FSR.Variable			:= Variable;
FSR.eReturnCode			:= eReturnCode;

// Forward to ITC
F_ITC_SendFSR := fbITC_Manager.M_SendData(
					meChannel	:= eChannelSrc,
					mMsgType	:= E_ITC_MsgTypeConv.FUNCTION_STATUS_REPORT,
					mpData		:= ADR(FSR),
					mLen		:= SIZEOF(FSR));

END_FUNCTION

// ---- 20_Product/10_BCF/11_Conv/11_Com/11_ITC/F_ITC_SendGVR.TcPOU
FUNCTION F_ITC_SendGVR : BOOL
(**************************************************************************************
 * 	Application		:	BoxControl Framework
 *	Revision		:	$Revision: 404529 $
 *	Revision date	:	$Date: 2018-04-23 08:21:38 +0200 (Mo., 23 Apr 2018) $
 *	Last changed by	:	$Author: b7bolm $
 *	URL				:	$URL: http://almscdc.swisslog.com/repo/SWPD/Development/BoxControlFramework/20_Release/trunk/01_Software/BCF/BCF/JumpStart/20_Product/10_App/11_Com/10_Lib/10_Conv/11_ITC/F_ITC_SendGVR.TcPOU $
 *
 *	Purpose			:	Wrap message - GVR
 *
 * ------------------------------------------------------------------------------------
 *	Copyright Swisslog [IP AG], Switzerland. All rights reserved.
 * 
 * ------------------------------------------------------------------------------------
 *	
 * 	Revision History: 
 *
 * 	VERSION			DATE			INITIALS			DESCRIPTION
 *	0.1				01.01.2001		swl					Example
 *
 **************************************************************************************)
VAR_INPUT
	eChannelSrc		: E_MFCS_Channel; // Source communicaton channel
	Number			: INT; // Number
	Quantity		: INT; // Quantity
	Variable0		: DINT; // Variable
	Variable1		: DINT; // Variable
	Variable2		: DINT; // Variable
	Variable3		: DINT; // Variable
	Variable4		: DINT; // Variable
	Variable5		: DINT; // Variable
	Variable6		: DINT; // Variable
	Variable7		: DINT; // Variable
	Variable8		: DINT; // Variable
	Variable9		: DINT; // Variable
	ReturnCode		: INT; // ReturnCode
END_VAR
VAR
	GVR					: ST_ITC_GVR; 
END_VAR

// Map values
GVR.Number := Number;
GVR.Quantity := Quantity;
GVR.Variable[0] := Variable0;
GVR.Variable[1] := Variable1;
GVR.Variable[2] := Variable2;
GVR.Variable[3] := Variable3;
GVR.Variable[4] := Variable4;
GVR.Variable[5] := Variable5;
GVR.Variable[6] := Variable6;
GVR.Variable[7] := Variable7;
GVR.Variable[8] := Variable8;
GVR.Variable[9] := Variable9;
GVR.ReturnCode := ReturnCode;

// Forward to ITC
F_ITC_SendGVR := fbITC_Manager.M_SendData(
					meChannel	:= eChannelSrc,
					mMsgType	:= E_ITC_MsgTypeConv.GLOBAL_VARIABLE_REPORT,
					mpData		:= ADR(GVR),
					mLen		:= SIZEOF(GVR));

END_FUNCTION

// ---- 20_Product/10_BCF/11_Conv/11_Com/11_ITC/F_ITC_SendIPR.TcPOU
FUNCTION F_ITC_SendIPR : BOOL
(**************************************************************************************
 * 	Application		:	BoxControl Framework
 *	Revision		:	$Revision: 404529 $
 *	Revision date	:	$Date: 2018-04-23 08:21:38 +0200 (Mo., 23 Apr 2018) $
 *	Last changed by	:	$Author: b7bolm $
 *	URL				:	$URL: http://almscdc.swisslog.com/repo/SWPD/Development/BoxControlFramework/20_Release/trunk/01_Software/BCF/BCF/JumpStart/20_Product/10_App/11_Com/10_Lib/10_Conv/11_ITC/F_ITC_SendIPR.TcPOU $
 *
 *	Purpose			:	Wrap message - IPR
 *
 * ------------------------------------------------------------------------------------
 *	Copyright Swisslog [IP AG], Switzerland. All rights reserved.
 * 
 * ------------------------------------------------------------------------------------
 *	
 * 	Revision History: 
 *
 * 	VERSION			DATE			INITIALS			DESCRIPTION
 *	0.1				01.01.2001		swl					Example
 *
 **************************************************************************************)
VAR_INPUT
	eChannelSrc			: E_MFCS_Channel; // Source communicaton channel
	Position			: STRING(Conveyor.POSITION_STRINGLENGTH); // SIS MM-GGG-EEEE-FF-Z
	TU_DataIndex		: DINT; // TU-DataIndex
	MSG_Sequence		: INT; // Assignment message sequence
	TU_ID				: STRING(Conveyor.TU_ID_STRINGLENGTH); // 18 Char SSID
	TU_Type				: INT; // TU-Type
	AssignmentID		: UDINT; // Assignment id
	Height				: INT; // Height Result
	WidthRight			: INT; // Width Right Result
	WidthLeft			: INT; // Width Left Result
	LengthFront			: INT; // Length Front Result
	LengthRear			: INT; // Length Rear Result
	Weight				: DINT; // Weight Value
	Tunnel				: INT; // Tunnel Result
	Runner				: INT; // Runner Result
	ErrorCode			: INT; // Error
	ValidLabelString	: INT; // Valid Label Return Code
	Label				: STRING(Conveyor.LABEL_LENGTH); // Characters of Label Data
END_VAR
VAR
	IPR					: ST_ITC_IPR; 
END_VAR

// Map values
IPR.Position := Position;
IPR.TU_DataIndex := TU_DataIndex;
IPR.MSG_Sequence := MSG_Sequence;
IPR.TU_ID := TU_ID;
IPR.TU_Type := TU_Type;
IPR.AssignmentID := AssignmentID;
IPR.Height := Height;
IPR.WidthRight := WidthRight;
IPR.WidthLeft := WidthLeft;
IPR.LengthFront := LengthFront;
IPR.LengthRear := LengthRear;
IPR.Weight := Weight;
IPR.Tunnel := Tunnel;
IPR.Runner := Runner;
IPR.ErrorCode := ErrorCode;
IPR.ValidLabelString := ValidLabelString;
IPR.Label := Label;

// Forward to ITC
F_ITC_SendIPR := fbITC_Manager.M_SendData(
					meChannel	:= eChannelSrc,
					mMsgType	:= E_ITC_MsgTypeConv.IDENTIFICATION_REPORT,
					mpData		:= ADR(IPR),
					mLen		:= SIZEOF(IPR));

END_FUNCTION

// ---- 20_Product/10_BCF/11_Conv/11_Com/11_ITC/F_ITC_SendISR.TcPOU
FUNCTION F_ITC_SendISR : BOOL
(**************************************************************************************
 * 	Application		:	BoxControl Framework
 *	Revision		:	$Revision: 404529 $
 *	Revision date	:	$Date: 2018-04-23 08:21:38 +0200 (Mo., 23 Apr 2018) $
 *	Last changed by	:	$Author: b7bolm $
 *	URL				:	$URL: http://almscdc.swisslog.com/repo/SWPD/Development/BoxControlFramework/20_Release/trunk/01_Software/BCF/BCF/JumpStart/20_Product/10_App/11_Com/10_Lib/10_Conv/11_ITC/F_ITC_SendISR.TcPOU $
 *
 *	Purpose			:	Wrap message - ISR
 *
 * ------------------------------------------------------------------------------------
 *	Copyright Swisslog [IP AG], Switzerland. All rights reserved.
 * 
 * ------------------------------------------------------------------------------------
 *	
 * 	Revision History: 
 *
 * 	VERSION			DATE			INITIALS			DESCRIPTION
 *	0.1				01.01.2001		swl					Example
 *
 **************************************************************************************)
VAR_INPUT
	eChannelSrc			: E_MFCS_Channel; // Source communicaton channel		
	SignalType			: INT; // Signal Type (0=Inputs, 1=Outputs, 2=Positions)
	StartSignalNumber	: INT; // Start Signal Number
	DataLength			: INT; // Data Length
	Information			: STRING(99); // (HEX) Information Data
	eReturnCode			: E_ErrorConv; // Return code
END_VAR
VAR
	ISR					: ST_ITC_ISR; 
END_VAR

// Map values
ISR.StartSignalNumber := StartSignalNumber;
ISR.SignalType := SignalType;
ISR.DataLength := DataLength;
ISR.Information := Information;
ISR.ReturnCode := eReturnCode;

// Forward to ITC
F_ITC_SendISR := fbITC_Manager.M_SendData(
					meChannel	:= eChannelSrc,
					mMsgType	:= E_ITC_MsgTypeConv.I_O_STATUS_REPORT,
					mpData		:= ADR(ISR),
					mLen		:= SIZEOF(ISR));

END_FUNCTION

// ---- 20_Product/10_BCF/11_Conv/11_Com/11_ITC/F_ITC_SendMCR.TcPOU
FUNCTION F_ITC_SendMCR : BOOL
(**************************************************************************************
 * 	Application		:	BoxControl Framework
 *	Revision		:	$Revision: 404529 $
 *	Revision date	:	$Date: 2018-04-23 08:21:38 +0200 (Mo., 23 Apr 2018) $
 *	Last changed by	:	$Author: b7bolm $
 *	URL				:	$URL: http://almscdc.swisslog.com/repo/SWPD/Development/BoxControlFramework/20_Release/trunk/01_Software/BCF/BCF/JumpStart/20_Product/10_App/11_Com/10_Lib/10_Conv/11_ITC/F_ITC_SendMCR.TcPOU $
 *
 *	Purpose			:	Wrap message - MCR
 *
 * ------------------------------------------------------------------------------------
 *	Copyright Swisslog [IP AG], Switzerland. All rights reserved.
 * 
 * ------------------------------------------------------------------------------------
 *	
 * 	Revision History: 
 *
 * 	VERSION			DATE			INITIALS			DESCRIPTION
 *	0.1				01.01.2001		swl					Example
 *
 **************************************************************************************)
VAR_INPUT
	eChannelSrc			: E_MFCS_Channel; // Source communicaton channel	
	Position			: STRING(Conveyor.POSITION_STRINGLENGTH); // Position
	Code				: INT; // Code
	Mode				: INT; // Mode
	Speed				: ST_ITC_ManualMotionSpeed; // Speed
	Axis				: ARRAY[1..6] OF ST_ITC_ManualMotionAxis; // Axis
	Button				: ARRAY[1..2] OF ST_ITC_ManualMotionSelection; // Buttons
	eReturnCode			: E_ErrorConv; // Return code
END_VAR
VAR
	MCR					: ST_ITC_MCR; 
END_VAR

// Map values
MCR.Position := Position;
MCR.Speed := Speed;
MCR.Mode := Mode;
MCR.Code := Code;
MCR.Axis := Axis;
MCR.Button := Button;
MCR.eReturnCode := eReturnCode;

// Forward to ITC
F_ITC_SendMCR := fbITC_Manager.M_SendData(
					meChannel	:= eChannelSrc,
					mMsgType	:= E_ITC_MsgTypeConv.MANUAL_CONTROL_REPORT,
					mpData		:= ADR(MCR),
					mLen		:= SIZEOF(MCR));

END_FUNCTION

// ---- 20_Product/10_BCF/11_Conv/11_Com/11_ITC/F_ITC_SendMSG.TcPOU
FUNCTION F_ITC_SendMSG : BOOL
(**************************************************************************************
 * 	Application		:	BoxControl Framework
 *	Revision		:	$Revision: 404529 $
 *	Revision date	:	$Date: 2018-04-23 08:21:38 +0200 (Mo., 23 Apr 2018) $
 *	Last changed by	:	$Author: b7bolm $
 *	URL				:	$URL: http://almscdc.swisslog.com/repo/SWPD/Development/BoxControlFramework/20_Release/trunk/01_Software/BCF/BCF/JumpStart/20_Product/10_App/11_Com/10_Lib/10_Conv/11_ITC/F_ITC_SendMSG.TcPOU $
 *
 *	Purpose			:	Sends customized MSG telegrams
 *
 * ------------------------------------------------------------------------------------
 *	Copyright Swisslog [IP AG], Switzerland. All rights reserved.
 * 
 * ------------------------------------------------------------------------------------
 *	
 * 	Revision History: 
 *
 * 	VERSION			DATE			INITIALS			DESCRIPTION
 *	0.1				01.01.2001		swl					Example
 *
 **************************************************************************************)
VAR_INPUT
	eChannelSrc		: E_MFCS_Channel; // Source communicaton channel	
	pMsgData		: PVOID; // Pointer to message structure
	Len				: UDINT; // Length of structure SIZEOF/LEN
END_VAR
VAR
	;
END_VAR


// Forward to ITC
F_ITC_SendMSG := fbITC_Manager.M_SendData(
					meChannel	:= eChannelSrc,
					mMsgType	:= E_ITC_MsgTypeConv.DATA_MESSAGE,
					mpData		:= pMsgData,
					mLen		:= Len);

END_FUNCTION

// ---- 20_Product/10_BCF/11_Conv/11_Com/11_ITC/F_ITC_SendPOR.TcPOU
FUNCTION F_ITC_SendPOR : BOOL
(**************************************************************************************
 * 	Application		:	BoxControl Framework
 *	Revision		:	$Revision: 404529 $
 *	Revision date	:	$Date: 2018-04-23 08:21:38 +0200 (Mo., 23 Apr 2018) $
 *	Last changed by	:	$Author: b7bolm $
 *	URL				:	$URL: http://almscdc.swisslog.com/repo/SWPD/Development/BoxControlFramework/20_Release/trunk/01_Software/BCF/BCF/JumpStart/20_Product/10_App/11_Com/10_Lib/10_Conv/11_ITC/F_ITC_SendPOR.TcPOU $
 *
 *	Purpose			:	Wrap message - POR
 *
 * ------------------------------------------------------------------------------------
 *	Copyright Swisslog [IP AG], Switzerland. All rights reserved.
 * 
 * ------------------------------------------------------------------------------------
 *	
 * 	Revision History: 
 *
 * 	VERSION			DATE			INITIALS			DESCRIPTION
 *	0.1				01.01.2001		swl					Example
 *
 **************************************************************************************)
VAR_INPUT
	eChannelSrc			: E_MFCS_Channel; // Source communicaton channel		
	Position			: STRING(Conveyor.POSITION_STRINGLENGTH); // SIS MM-GGG-EEEE-FF-Z
	TU_ID				: STRING(Conveyor.TU_ID_STRINGLENGTH); // 18 Digit SSID
	TU_Type				: INT; // TU Type
	AssignmentID		: UDINT; // assignment id
	LoadInformation		: BOOL; // Load Information
END_VAR
VAR
	POR				: ST_ITC_POR; 
END_VAR

// Map values
POR.Position := Position;
POR.AssignmentID := AssignmentID;
POR.LoadInformation := LoadInformation;
POR.TU_ID := TU_ID;
POR.TU_Type := TU_Type;

// Forward to ITC
F_ITC_SendPOR := fbITC_Manager.M_SendData(
					meChannel	:= eChannelSrc,
					mMsgType	:= E_ITC_MsgTypeConv.POSITION_OCCUPIED_REPORT,
					mpData		:= ADR(POR),
					mLen		:= SIZEOF(POR));

END_FUNCTION

// ---- 20_Product/10_BCF/11_Conv/11_Com/11_ITC/F_ITC_SendRAC.TcPOU
FUNCTION F_ITC_SendRAC : BOOL
(**************************************************************************************
 * 	Application		:	BoxControl Framework
 *	Revision		:	$Revision: 404529 $
 *	Revision date	:	$Date: 2018-04-23 08:21:38 +0200 (Mo., 23 Apr 2018) $
 *	Last changed by	:	$Author: b7bolm $
 *	URL				:	$URL: http://almscdc.swisslog.com/repo/SWPD/Development/BoxControlFramework/20_Release/trunk/01_Software/BCF/BCF/JumpStart/20_Product/10_App/11_Com/10_Lib/10_Conv/11_ITC/F_ITC_SendRAC.TcPOU $
 *
 *	Purpose			:	Wrap message - RAC
 *
 * ------------------------------------------------------------------------------------
 *	Copyright Swisslog [IP AG], Switzerland. All rights reserved.
 * 
 * ------------------------------------------------------------------------------------
 *	
 * 	Revision History: 
 *
 * 	VERSION			DATE			INITIALS			DESCRIPTION
 *	0.1				01.01.2001		swl					Example
 *
 **************************************************************************************)
VAR_INPUT
	eChannelSrc				: E_MFCS_Channel; // Source communicaton channel
	PositionName			: STRING(Conveyor.POSITION_STRINGLENGTH); // SIS MM-GGG-EEEE-FF-Z
	CommandDataIndex		: INT;
	AssignmentID			: UDINT;
	GroupID					: ULINT;
	eReturnCode				: E_ErrorConv; // Return code
END_VAR
VAR
	RAC						: ST_ITC_RAC; 
END_VAR

// Map values
RAC.Position := PositionName;
RAC.CommandDataIndex := CommandDataIndex;
RAC.AssignmentID := AssignmentID;
RAC.GroupID := GroupID;
RAC.eReturnCode := eReturnCode;

// Forward to ITC
F_ITC_SendRAC := fbITC_Manager.M_SendData(
					meChannel	:= eChannelSrc,
					mMsgType	:= E_ITC_MsgTypeConv.ROBOT_ACTION_COMPLETE,
					mpData		:= ADR(RAC),
					mLen		:= SIZEOF(RAC));

END_FUNCTION

// ---- 20_Product/10_BCF/11_Conv/11_Com/11_ITC/F_ITC_SendRAQ.TcPOU
FUNCTION F_ITC_SendRAQ : BOOL
(**************************************************************************************
 * 	Application		:	BoxControl Framework
 *	Revision		:	$Revision: 404529 $
 *	Revision date	:	$Date: 2018-04-23 08:21:38 +0200 (Mo., 23 Apr 2018) $
 *	Last changed by	:	$Author: b7bolm $
 *	URL				:	$URL: http://almscdc.swisslog.com/repo/SWPD/Development/BoxControlFramework/20_Release/trunk/01_Software/BCF/BCF/JumpStart/20_Product/10_App/11_Com/10_Lib/10_Conv/11_ITC/F_ITC_SendRAQ.TcPOU $
 *
 *	Purpose			:	Wrap message - RAQ
 *
 * ------------------------------------------------------------------------------------
 *	Copyright Swisslog [IP AG], Switzerland. All rights reserved.
 * 
 * ------------------------------------------------------------------------------------
 *	
 * 	Revision History: 
 *
 * 	VERSION			DATE			INITIALS			DESCRIPTION
 *	0.1				01.01.2001		swl					Example
 *
 **************************************************************************************)
VAR_INPUT
	eChannelSrc				: E_MFCS_Channel; // Source communicaton channel
	PositionName			: STRING(Conveyor.POSITION_STRINGLENGTH); // SIS MM-GGG-EEEE-FF-Z
	GroupID					: ULINT;
	NumberOfRA				: INT;
END_VAR
VAR
	RAQ						: ST_ITC_RAQ; 
END_VAR

// Map values
RAQ.Position := PositionName;
RAQ.GroupID := GroupID;
RAQ.NumberOfRA := NumberOfRA;

// Forward to ITC
F_ITC_SendRAQ := fbITC_Manager.M_SendData(
					meChannel	:= eChannelSrc,
					mMsgType	:= E_ITC_MsgTypeConv.ROBOT_ACTION_REQUEST,
					mpData		:= ADR(RAQ),
					mLen		:= SIZEOF(RAQ));

END_FUNCTION

// ---- 20_Product/10_BCF/11_Conv/11_Com/11_ITC/F_ITC_SendRDR.TcPOU
FUNCTION F_ITC_SendRDR : BOOL
(**************************************************************************************
 * 	Application		:	BoxControl Framework
 *	Revision		:	$Revision: 404529 $
 *	Revision date	:	$Date: 2018-04-23 08:21:38 +0200 (Mo., 23 Apr 2018) $
 *	Last changed by	:	$Author: b7bolm $
 *	URL				:	$URL: http://almscdc.swisslog.com/repo/SWPD/Development/BoxControlFramework/20_Release/trunk/01_Software/BCF/BCF/JumpStart/20_Product/10_App/11_Com/10_Lib/10_Conv/11_ITC/F_ITC_SendRDR.TcPOU $
 *
 *	Purpose			:	Wrap message - RDR
 *
 * ------------------------------------------------------------------------------------
 *	Copyright Swisslog [IP AG], Switzerland. All rights reserved.
 * 
 * ------------------------------------------------------------------------------------
 *	
 * 	Revision History: 
 *
 * 	VERSION			DATE			INITIALS			DESCRIPTION
 *	0.1				01.01.2001		swl					Example
 *
 **************************************************************************************)
VAR_INPUT
	eChannelSrc			: E_MFCS_Channel; // Source communicaton channel
	PositionName		: STRING(Conveyor.POSITION_STRINGLENGTH); // SIS MM-GGG-EEEE-FF-Z
	CommandDataIndex	: DINT;
	AssignmentID		: UDINT; // assignment id
	GroupID				: ULINT;
	eReturnCode			: E_ErrorConv; // Return code
END_VAR
VAR
	RDR				: ST_ITC_RDR; 
END_VAR

// Map values
RDR.Position := PositionName;
RDR.CommandDataIndex := CommandDataIndex;
RDR.AssignmentID := AssignmentID;
RDR.GroupID := GroupID;
RDR.ReturnCode := eReturnCode;

// Forward to ITC
F_ITC_SendRDR := fbITC_Manager.M_SendData(
					meChannel	:= eChannelSrc,
					mMsgType	:= E_ITC_MsgTypeConv.ROBOT_DELETE_REPORT,
					mpData		:= ADR(RDR),
					mLen		:= SIZEOF(RDR));

END_FUNCTION

// ---- 20_Product/10_BCF/11_Conv/11_Com/11_ITC/F_ITC_SendSIR.TcPOU
FUNCTION F_ITC_SendSIR : BOOL
(**************************************************************************************
 * 	Application		:	BoxControl Framework
 *	Revision		:	$Revision: 404529 $
 *	Revision date	:	$Date: 2018-04-23 08:21:38 +0200 (Mo., 23 Apr 2018) $
 *	Last changed by	:	$Author: b7bolm $
 *	URL				:	$URL: http://almscdc.swisslog.com/repo/SWPD/Development/BoxControlFramework/20_Release/trunk/01_Software/BCF/BCF/JumpStart/20_Product/10_App/11_Com/10_Lib/10_Conv/11_ITC/F_ITC_SendSIR.TcPOU $
 *
 *	Purpose			:	Wrap message - SIR
 *
 * ------------------------------------------------------------------------------------
 *	Copyright Swisslog [IP AG], Switzerland. All rights reserved.
 * 
 * ------------------------------------------------------------------------------------
 *	
 * 	Revision History: 
 *
 * 	VERSION			DATE			INITIALS			DESCRIPTION
 *	0.1				01.01.2001		swl					Example
 *
 **************************************************************************************)
VAR_INPUT
	eChannelSrc		: E_MFCS_Channel; // Source communicaton channel	
	PositionName	: STRING(Conveyor.POSITION_STRINGLENGTH); // SIS MM-GGG-EEEE-FF-Z
	Code			: INT; // Code
	TU_ID			: STRING(Conveyor.TU_ID_STRINGLENGTH); // 18 Digit SSID
	Counter1		: DINT; // Counter 1
	Counter2		: DINT; // Counter 2
	Counter3		: DINT; // Counter 3
	Counter4		: DINT; // Counter 4
	Counter5		: DINT; // Counter 5
	eReturnCode		: E_ErrorConv; // Return code
END_VAR
VAR
	SIR				: ST_ITC_SIR; 
END_VAR

